Yaskawa INFORM job: OK_R2_O57-69(2)(90,0)_OK_HARDOX.JBI

/JOB
//NAME OK_R2_O57-69(2)(90,0)_OK_HARDOX
///FOLDERNAME X4
//POS
///NPOS 604,604,604,23,0,0
///TOOL 0
///POSTYPE PULSE
///PULSE
C00000=-135424,72899,29147,-3537,85342,3792
C00001=-134013,95021,61136,-4029,77105,4505
C00002=-134047,101087,71818,-4077,73656,4607
C00003=-134047,101216,72822,-4088,73105,4626
C00004=-134047,101094,71866,-4078,73630,4609
C00005=-133936,105187,77198,-4137,72460,4688
C00006=-134047,101094,71866,-4078,73630,4609
C00007=-133891,92563,58880,-4064,77236,4542
C00008=-133627,85963,47659,-4101,80754,4516
C00009=-133192,78294,50454,-10127,76922,11696
C00010=-133849,85255,61933,-10093,73405,11757
C00011=-135353,87618,67605,-9788,70974,11422
C00012=-135353,87997,69106,-9827,70255,11481
C00013=-135353,87618,67605,-9788,70974,11422
C00014=-135153,93739,75342,-9940,69404,11624
C00015=-135353,87618,67605,-9788,70974,11422
C00016=-133639,83161,60388,-10158,73308,11840
C00017=-132974,76301,49087,-10194,76769,11784
C00018=-129415,62996,33414,-11066,79991,12732
C00019=-98130,32671,61537,-45409,44339,32891
C00020=-100023,41688,73231,-46965,41628,33506
C00021=-100756,49088,84228,-49401,39255,34803
C00022=-100756,52120,89278,-50881,38240,35655
C00023=-100756,49088,84228,-49401,39255,34803
C00024=-101219,51120,86580,-49709,38764,34882
C00025=-100756,49088,84228,-49401,39255,34803
C00026=-97195,31965,62320,-46227,44186,33575
C00027=-75566,-2034,22500,-42402,86688,50389
C00028=-92276,-18388,7402,-33699,73725,46550
C00029=-92276,-17400,9548,-33822,73042,46763
C00030=-92276,-17933,8393,-33755,73407,46648
C00031=-120131,-32698,-12117,4829,66200,34356
C00032=-120131,-32114,-10702,4851,65630,34332
C00033=-120989,-32117,-10704,5006,65680,34020
C00034=-120131,-32114,-10702,4851,65630,34332
C00035=-120131,-38085,-26806,4645,72450,34604
C00036=-99101,-76935,-92016,-31014,74911,20401
C00037=-52587,-144740,-101483,-60524,64363,-65274
C00038=-46989,-65360,-59229,-62781,73103,-77672
C00039=-56832,-65466,-56421,-59287,64983,-77772
C00040=-57148,-65688,-55453,-59188,64110,-77279
C00041=-55649,-62097,-53047,-61106,66880,-78547
C00042=-57237,-59710,-51792,-60669,66110,-79037
C00043=-56277,-61326,-53166,-60831,66721,-78866
C00044=-55441,-62561,-53810,-61057,67127,-78609
C00045=-56207,-63985,-54541,-61032,66503,-78630
C00046=-55438,-62578,-53813,-61060,67126,-78606
C00047=-51973,-62323,-54701,-62406,69323,-78001
C00048=-48054,-62529,-57040,-62601,72472,-77896
C00049=-29811,-70761,-60283,-66780,94863,-53671
C00050=-30965,-22538,-31531,-67696,97011,-56857
C00051=-55044,-42598,-44870,-68563,88788,-43678
C00052=-56249,-45120,-46406,-68472,87844,-43687
C00053=-57925,-45354,-44812,-68371,86292,-43442
C00054=-57925,-45174,-43802,-68390,86084,-43215
C00055=-57925,-45354,-44812,-68371,86292,-43442
C00056=-59167,-45210,-44726,-68282,85469,-43617
C00057=-57925,-45354,-44812,-68371,86292,-43442
C00058=-55819,-44223,-45863,-68504,88181,-43684
C00059=-44722,-31045,-43816,-69927,97696,-44632
C00060=-43071,-26445,-40665,-70170,98951,-44614
C00061=-127706,-49493,-81773,19458,97242,-49666
C00062=-127020,6423,-39070,7004,99714,-51816
C00063=-127020,5137,-37554,6966,98131,-51906
C00064=-128416,4382,-35850,7239,96821,-52416
C00065=-128416,3847,-35017,7224,96041,-52460
C00066=-128416,4148,-35496,7233,96488,-52435
C00067=-130041,4566,-35136,7580,96617,-52937
C00068=-129924,4205,-34639,7545,96120,-52933
C00069=-129457,4078,-34747,7447,96082,-52788
C00070=-130190,4712,-35256,7614,96778,-52976
C00071=-128966,36168,-17458,7491,101844,-52285
C00072=-149392,-6912,-25974,9982,75562,-31317
C00073=-149173,-488,-12666,10148,70714,-31647
C00074=-149173,-326,-10897,10208,69722,-31733
C00075=-149173,-394,-11578,10184,70101,-31701
C00076=-148123,2416,-9216,9823,69962,-31333
C00077=-149173,-394,-11578,10184,70101,-31701
C00078=-152478,4885,-6741,15795,72623,-37698
C00079=-151455,3828,-7649,15488,72442,-37350
C00080=-152478,4560,-12614,15554,75946,-37261
C00081=-146445,-24647,-43161,13522,78564,-34847
C00082=-131268,-45047,-56509,8633,74300,53297
C00083=-142507,25021,6402,32310,105830,54923
C00084=-142507,25105,7931,32155,105064,54695
C00085=-142507,25067,7336,32214,105361,54783
C00086=-144899,27115,9325,31955,106116,54020
C00087=-144899,27165,10051,31882,105756,53914
C00088=-143964,26333,9240,31989,105467,54213
C00089=-144899,27115,9325,31955,106116,54020
C00090=-139799,26044,8286,32411,104272,55572
C00091=-139799,26086,8928,32350,103953,55476
C00092=-140218,24332,7231,32337,104232,55386
C00093=-139845,24485,5469,32557,105080,55794
C00094=-133821,6451,-11055,33047,103540,57803
C00095=-133821,6495,-9064,32866,102523,57496
C00096=-133821,6476,-9598,32913,102793,57577
C00097=-132525,9567,-6887,32955,102227,57935
C00098=-132525,9588,-6343,32910,101953,57853
C00099=-133066,7796,-7920,32894,102203,57708
C00100=-133013,8554,-8607,33013,102871,57931
C00101=-134496,-11545,-24055,37394,79049,50318
C00102=-128731,-14923,-26642,36062,76491,51870
C00103=-127482,-15460,-24018,36014,74425,51702
C00104=-127482,-15304,-22595,36136,73774,51482
C00105=-127482,-15363,-23111,36090,74009,51562
C00106=-129060,-19650,-26295,36507,74476,51047
C00107=-129060,-19568,-25628,36564,74177,50944
C00108=-128523,-17977,-24457,36422,74028,51123
C00109=-129540,-19245,-27224,36505,75313,51130
C00110=-136115,2071,-10391,37882,78617,49479
C00111=-137580,2242,-9921,38197,79097,49024
C00112=-137580,2375,-8533,38282,78470,48799
C00113=-137580,2298,-9294,38235,78811,48922
C00114=-139070,-1458,-12440,38519,79473,48520
C00115=-139070,-1365,-11538,38571,79071,48374
C00116=-138460,140,-10285,38458,78803,48541
C00117=-138988,-820,-13903,38388,80409,48895
C00118=-141740,13451,-1511,38926,81398,48075
C00119=-142514,14144,562,39136,81023,47605
C00120=-142514,14274,1799,39195,80477,47404
C00121=-142514,14207,1180,39164,80748,47504
C00122=-144026,10774,-1912,39404,81538,47142
C00123=-144026,10851,-1183,39436,81218,47023
C00124=-143517,12181,9,39358,80948,47144
C00125=-143717,11422,-2918,39282,82143,47501
C00126=-140568,19291,1223,17454,68729,44783
C00127=-141248,20501,3331,17792,68230,44452
C00128=-141248,20564,4327,17861,67675,44366
C00129=-141248,20543,3999,17838,67857,44394
C00130=-142986,16313,57,18468,68479,43839
C00131=-142986,16348,619,18508,68167,43788
C00132=-142176,18240,2371,18214,67887,44048
C00133=-142876,17282,-1215,18280,69673,44071
C00134=-131494,-80468,-98534,7816,92108,-53678
C00135=-52065,-14099,-27709,-42253,108676,27596
C00136=-76671,-130461,-121705,-35735,90710,50834
C00137=-94829,-93442,-100428,-28991,96183,47377
C00138=-110716,-92055,-82664,-19311,98038,51285
C00139=-114275,-93352,-80055,-19461,95045,50478
C00140=-118122,-92212,-76367,-19656,92534,49497
C00141=-118129,-91398,-74848,-19645,92046,49575
C00142=-118122,-92212,-76367,-19656,92534,49497
C00143=-119808,-92271,-76389,-19753,92113,48959
C00144=-118122,-92212,-76367,-19656,92534,49497
C00145=-114499,-91094,-78376,-19482,95112,50387
C00146=-110992,-89821,-80983,-19339,98080,51178
C00147=-124454,-89651,-86550,11137,94998,-69701
C00148=-122569,-92184,-83910,11067,91866,-69331
C00149=-120652,-93960,-80852,11027,88857,-68936
C00150=-120652,-93520,-79457,11027,88237,-68992
C00151=-120652,-93960,-80852,11027,88857,-68936
C00152=-120650,-97396,-81866,11026,87737,-69033
C00153=-120652,-93960,-80852,11027,88857,-68936
C00154=-118161,-93768,-80427,10994,88357,-68121
C00155=-120652,-93960,-80852,11027,88857,-68936
C00156=-120037,-91891,-82714,11032,90945,-68539
C00157=-121981,-89592,-85452,11099,94026,-68936
C00158=-122005,-89480,-97857,11363,101580,-68254
C00159=-122005,-89427,-98101,11372,101754,-68238
C00160=-119094,-95812,-115555,-4544,90851,-20867
C00161=-116502,-111480,-109655,-18779,62868,21987
C00162=-119472,-101923,-104261,-17094,63743,20698
C00163=-121534,-96097,-100090,-16016,63743,19914
C00164=-121534,-96194,-98882,-16123,62979,20025
C00165=-112336,-84014,-94514,-26506,72534,27449
C00166=-114298,-84401,-94682,-25743,71847,26864
C00167=-121534,-96097,-100090,-16016,63743,19914
C00168=-121514,-92242,-98700,-15883,64832,19765
C00169=-121534,-96097,-100090,-16016,63743,19914
C00170=-119823,-101836,-103002,-17025,62972,20682
C00171=-116876,-111303,-108368,-18711,62117,21969
C00172=-126032,-109701,-108999,21760,66785,-27050
C00173=-122513,-101468,-103921,20079,66940,-25677
C00174=-121483,-94377,-99419,19507,67520,-25186
C00175=-121483,-94509,-98158,19621,66724,-25324
C00176=-121483,-94377,-99419,19507,67520,-25186
C00177=-119206,-94355,-99408,18489,67008,-24418
C00178=-121483,-94377,-99419,19507,67520,-25186
C00179=-121468,-91005,-98354,19362,68535,-25006
C00180=-121483,-94377,-99419,19507,67520,-25186
C00181=-124810,-108862,-107603,21303,66070,-26716
C00182=-126981,-112864,-109311,24940,61360,-29729
C00183=-123200,-104180,-104415,22777,61614,-28126
C00184=-121230,-90686,-98732,21152,64298,-26805
C00185=-121230,-90968,-97120,21351,63235,-27013
C00186=-121230,-90806,-98119,21226,63888,-26884
C00187=-118688,-90754,-98099,19926,63280,-26013
C00188=-121230,-90721,-98563,21173,64184,-26826
C00189=-121211,-84894,-96124,20922,65577,-26553
C00190=-121230,-90686,-98732,21152,64298,-26805
C00191=-121413,-93580,-100796,21282,64141,-26906
C00192=-124847,-101623,-105736,23178,64029,-28268
C00193=-120616,-95755,-103879,23668,64726,-45447
C00194=-120621,-89459,-99052,23623,64971,-45396
C00195=-102398,-78806,-99215,-137,71874,-40792
C00196=-120614,-97387,-102466,23992,63157,-45792
C00197=-122354,-96256,-100860,24938,63287,-46459
C00198=-99477,-102621,-105563,-1650,63574,-39713
C00199=-93449,-138180,-112622,-5538,49931,-36849
C00200=-85999,-163182,-115201,-11989,39587,-32297
C00201=-96470,-180165,-126119,-4784,36529,-37522
C00202=-120616,-95173,-105764,23303,89544,-42444
C00203=-107191,-96001,-89285,21702,28532,-58770
C00204=-107187,-93630,-79997,25295,24388,-60561
C00205=-107188,-92928,-77886,26213,23539,-61010
C00206=-112362,-77289,-77026,28293,40281,-63318
C00207=-107081,-94020,-78768,26067,23489,-60939
C00208=-108911,-93070,-77209,29349,23678,-62538
C00209=-100555,-91608,-91171,7273,48196,-53989
C00210=-102645,-104114,-96524,14611,51707,-64227
C00211=-108915,-55552,-83371,19664,91458,-62056
C00212=-110657,-50226,-86705,20295,96355,-61815
C00213=-107202,-93991,-108886,21178,109925,-43661
C00214=-120660,-73953,-111348,177,99224,835
C00215=-120616,-96234,-101081,-23944,56754,46777
C00216=-120615,-96493,-97034,-24670,54353,47364
C00217=-120614,-96447,-94923,-25055,53191,47662
C00218=-125343,-63714,-87611,-17170,75461,41479
C00219=-118876,-96360,-94049,-26267,53277,48431
C00220=-120612,-97621,-95709,-25094,53083,47691
C00221=-124024,-105215,-109245,-22308,82546,38090
C00222=-123496,-104488,-108175,-22872,85665,42107
C00223=-120617,-94319,-107453,-23464,90858,42123
C00224=-120617,-92878,-109780,-23521,92858,41729
C00225=-120619,-86141,-115603,-23930,99335,40429
C00226=-120619,-89012,-115558,8782,73464,77384
C00227=-120618,-92353,-112869,8941,70132,77138
C00228=-120618,-93422,-111698,9011,68877,77043
C00229=-120616,-94109,-113157,8979,69414,77085
C00230=-120318,-89311,-110489,8778,70198,77244
C00231=-120618,-93688,-111329,9132,68044,76969
C00232=-120618,-93957,-110924,9216,67187,76884
C00233=-120618,-94299,-110440,9161,65769,76809
C00234=-120618,-94831,-109599,8469,63241,76696
C00235=-120617,-95145,-109027,7071,61401,76664
C00236=-120617,-95217,-108863,5672,60665,76701
C00237=-120618,-93036,-111930,4923,63538,76718
C00238=-120618,-92960,-112001,4009,63579,76743
C00239=-120618,-92691,-112274,2433,64167,76800
C00240=-120618,-92166,-112798,840,65602,76863
C00241=-120618,-91419,-113490,-342,67708,76910
C00242=-120619,-90739,-114068,-878,69589,76936
C00243=-120619,-89701,-115007,-939,71612,76812
C00244=-120619,-88814,-115609,-873,73870,76855
C00245=-120619,-87740,-116270,-151,76574,76959
C00246=-120619,-86987,-116700,1182,78540,77121
C00247=-120619,-86782,-116823,2462,79296,77267
C00248=-120619,-90672,-114378,3278,75949,77117
C00249=-120619,-90769,-114313,4130,75889,77177
C00250=-120619,-91109,-114056,5597,75252,77256
C00251=-120618,-91719,-113544,7101,73764,77286
C00252=-120618,-92472,-112836,8259,71637,77242
C00253=-120618,-92872,-112418,8666,70405,77193
C00254=-120618,-93168,-112034,8862,69621,77111
C00255=-120618,-93422,-111698,9011,68877,77043
C00256=-120618,-92353,-112869,8941,70132,77138
C00257=-120619,-89012,-115558,8782,73464,77384
C00258=-120595,-119438,-127420,-8829,91162,8830
C00259=-129025,-103888,-99333,21372,86937,-54976
C00260=-120613,-94952,-86848,20336,81911,-52813
C00261=-120613,-94069,-83278,20415,80272,-53091
C00262=-106596,-117430,-87528,9818,57368,-33279
C00263=-120519,-95091,-83551,20421,79912,-53118
C00264=-122104,-92396,-81537,20633,80446,-53604
C00265=-112247,-111615,-87090,12951,66121,-41348
C00266=-120242,-93380,-81431,16167,85346,-56835
C00267=-120729,-92389,-78218,16226,84033,-57178
C00268=-121550,-94001,-78799,15119,86025,-61641
C00269=-122325,-96218,-79481,13215,89152,-68718
C00270=-120612,-93818,-82398,13271,91824,-67835
C00271=-120613,-94827,-86367,13308,93699,-67633
C00272=-120614,-96085,-95173,13466,98348,-67128
C00273=-120625,-105302,-100360,13404,96846,-67297
C00274=-102872,-120945,-93289,-41313,52454,35552
C00275=-111052,-89986,-73102,-36259,51528,31574
C00276=-114360,-89865,-71590,-35102,49434,30694
C00277=-117529,-82976,-67958,-32873,49251,29097
C00278=-113966,-89555,-70876,-35431,49366,30932
C00279=-115650,-91167,-72721,-34446,48930,30213
C00280=-116153,-87173,-73787,-30474,57370,33009
C00281=-115134,-90585,-78921,-28213,65812,37618
C00282=-114816,-93273,-83340,-25850,75230,43378
C00283=-115191,-85090,-71836,-25015,76673,46996
C00284=-114907,-96450,-75026,-24463,77444,52852
C00285=-115702,-94689,-74701,-23512,87260,62633
C00286=-112822,-91718,-77371,-23458,91001,62960
C00287=-109330,-92095,-80656,-23399,93677,63722
C00288=-110759,-94815,-97268,-24043,101385,61640
C00289=-25230,-87703,-86789,-41333,106155,-71905
C00290=-55862,19660,17206,-68346,89547,-53836
C00291=-59225,37567,25812,-69215,105770,-42705
C00292=-67658,42850,42597,-68102,97125,-40508
C00293=-69543,42635,44538,-68129,95346,-40204
C00294=-67599,42910,43858,-67984,96867,-40179
C00295=-68366,42138,41747,-68199,96713,-40671
C00296=-69537,42554,44453,-68130,95355,-40208
C00297=-69167,26414,28126,-68889,91591,-41841
C00298=-69430,8343,11443,-69273,87154,-43187
C00299=-70467,-11089,-4532,-69437,78929,-44678
C00300=-70464,-3151,1747,-68553,83829,-57137
C00301=-68177,-4212,-1280,-68454,85880,-57398
C00302=-65815,-3605,-3490,-68417,88124,-57797
C00303=-46513,-27715,-22241,-69125,80479,-38621
C00304=-7625,-19791,-74194,-84461,116832,-51132
C00305=-98528,-26744,-48644,-33463,55012,-18344
C00306=-113253,15209,27106,-3834,50657,3406
C00307=-113409,21623,32322,-3755,50736,3338
C00308=-112510,30954,47444,-4478,46281,3921
C00309=-113472,24070,39362,-3899,47665,3430
C00310=-113579,25546,39455,-3805,48359,3355
C00311=-112547,30896,47385,-4459,46286,3903
C00312=-113092,30984,47541,-6567,46499,5785
C00313=-107982,35826,53096,-19952,49307,15286
C00314=-107346,38752,56151,-24065,51859,19797
C00315=-102444,58818,79888,-34511,57818,35075
C00316=-101044,76619,103296,-39601,59307,41475
C00317=-99948,73081,91706,-37976,69105,42304
C00318=-99205,63215,84174,-37575,62603,39615
C00319=-97180,56339,73463,-36771,65900,39269
C00320=-108272,10166,23438,-3323,45242,19316
C00321=-109103,10218,12469,-2549,51979,18742
C00322=-99879,30934,32617,-21980,59339,34187
C00323=-99785,30090,30578,-21838,60128,34061
C00324=-99052,29053,30612,-22206,59809,34434
C00325=-101543,26260,28122,-21325,59243,33514
C00326=-98482,32149,35009,-29284,63220,41247
C00327=-92009,66840,89116,-42947,61850,57046
C00328=-89877,62120,80876,-42077,64804,56709
C00329=-70258,15873,38394,-48666,102593,69187
C00330=-68816,9929,45318,-53577,93501,68972
C00331=-74323,28982,63484,-55349,89726,68465
C00332=-74758,1474,21309,-45746,90270,65676
C00333=-98607,12568,39814,52966,86937,78252
C00334=-98596,22842,59344,53301,82774,75788
C00335=-96296,21421,60413,54092,80731,75703
C00336=-95348,20952,60953,54433,79893,75663
C00337=-96117,19164,58324,54129,80713,75783
C00338=-95662,23434,63388,54370,79922,75521
C00339=-95503,21312,61702,54422,79811,75531
C00340=-92574,18445,54645,48983,79889,68258
C00341=-91800,17848,53101,47601,79897,67557
C00342=-92530,17999,51917,47342,80806,67673
C00343=-94302,18640,49262,46764,83033,67943
C00344=-79003,18324,29303,31626,94586,4503
C00345=-64136,40618,57122,29721,84915,83830
C00346=-62802,39067,58740,29997,82892,83805
C00347=-62255,38544,59506,30121,82059,83791
C00348=-62254,37103,56589,30066,82978,84033
C00349=-62821,40643,61741,30049,81995,83562
C00350=-59984,48909,70165,26795,84201,83115
C00351=-59410,69261,96131,25367,86084,74959
C00352=-59404,69357,96256,25356,86081,74939
C00353=-59713,70793,96681,25260,86600,74945
C00354=-60461,74839,98386,25037,87745,74932
C00355=-60470,59585,70460,25309,96249,76737
C00356=-66845,10330,41939,25249,64720,33768
C00357=-66816,16396,52426,25952,61688,33052
C00358=-66804,19142,57057,26292,60387,32730
C00359=-66058,20615,58344,26298,60142,32956
C00360=-66868,17219,53699,26035,61378,32955
C00361=-66973,19658,57552,26302,60399,32669
C00362=-66985,16895,52895,25961,61707,32992
C00363=-67015,10800,42362,25255,64752,33711
C00364=-98181,31350,57269,53093,86032,77938
C00365=-96082,29267,57446,53647,84171,77916
C00366=-95219,28523,57622,53885,83405,77901
C00367=-95917,26905,55160,53675,84199,78019
C00368=-95506,31088,60230,53837,83386,77740
C00369=-95359,28788,58259,53869,83329,77779
C00370=-92697,26913,52373,48450,83827,70215
C00371=-91994,26523,51069,47073,83939,69440
C00372=-92656,26997,50292,46905,84772,69532
C00373=-94270,28412,48618,46533,86809,69749
C00374=-79891,40483,43632,25605,98381,-17488
C00375=-64421,55368,61348,15926,95442,-62339
C00376=-63205,52871,61672,16144,93779,-62133
C00377=-62708,51961,61917,16235,93087,-62052
C00378=-62707,50761,59239,16263,94078,-61920
C00379=-63223,54241,64482,16113,92796,-62269
C00380=-60236,62044,73663,12795,94061,-63101
C00381=-59090,69141,83012,10500,94867,-70833
C00382=-59083,69182,83067,10487,94869,-70851
C00383=-59379,71028,84054,10408,95242,-70919
C00384=-60098,76023,87068,10213,96031,-71094
C00385=-60107,66003,66038,10511,103704,-70448
C00386=-66860,35146,61423,22993,49349,53528
C00387=-66834,42827,74568,24499,45535,52525
C00388=-66824,46660,80883,25305,43786,52015
C00389=-66175,48781,83167,25255,43321,52183
C00390=-66880,43946,76304,24713,45097,52378
C00391=-66970,47398,81721,25407,43702,51920
C00392=-66981,43500,75311,24586,45473,52438
C00393=-67007,35727,62031,23060,49318,53454
C00394=-87565,40229,55167,37616,76398,68031
C00395=-104252,61764,84947,51561,88394,76219
C00396=-102517,58043,82852,52038,87086,76344
C00397=-101804,56689,82195,52237,86527,76380
C00398=-102435,54601,78919,52052,87454,76595
C00399=-101993,60636,86873,52209,86091,76036
C00400=-101932,57147,83104,52210,86393,76238
C00401=-99529,53434,74771,46937,87155,68655
C00402=-98895,52660,72970,45595,87312,67859
C00403=-99433,53501,72680,45467,88010,67934
C00404=-100745,55861,72292,45181,89689,68100
C00405=-89942,52639,54543,22757,100290,-22350
C00406=-84530,60242,66965,10989,97828,-69052
C00407=-83700,56528,65849,11170,96516,-68885
C00408=-83359,55133,65530,11245,95959,-68819
C00409=-83358,53843,62725,11276,97003,-68723
C00410=-83705,58033,68848,11139,95464,-68982
C00411=-80399,62193,73871,7256,96460,-69699
C00412=-78998,67441,80988,4366,97017,-77318
C00413=-78990,67470,81028,4351,97018,-77335
C00414=-79114,69587,82331,4315,97310,-77366
C00415=-79414,75293,86196,4226,97877,-77446
C00416=-79422,65472,65446,4368,105580,-77179
C00417=-80352,27457,54566,26195,53383,48637
C00418=-80356,27473,54581,26196,53382,48635
C00419=-80357,27479,54587,26196,53382,48634
C00420=-79589,28666,55655,26054,53112,48894
C00421=-80424,25883,51570,25884,54338,48863
C00422=-80357,27479,54587,26196,53382,48634
C00423=-80356,27473,54581,26196,53382,48635
C00424=-80352,27458,54566,26195,53383,48637
C00425=-110061,-17560,-36552,26636,92274,45980
C00426=-111839,-83491,-103870,27371,99587,47031
C00427=-38426,-40229,-52385,-46753,77455,-20722
C00428=-20805,-37224,-43776,-64442,70782,-24410
C00429=-53615,-60479,-29767,-71413,48188,-35364
C00430=-53622,-60473,-29764,-71411,48184,-35366
C00431=-53625,-60471,-29763,-71411,48182,-35366
C00432=-52450,-61746,-30400,-71683,48877,-35041
C00433=-53622,-61330,-31549,-70858,48414,-35743
C00434=-53667,-60425,-29740,-73440,59962,-39458
C00435=-53705,-60384,-29719,-74506,70698,-55233
C00436=-53706,-60382,-29718,-74560,71274,-55582
C00437=-53707,-60381,-29717,-74560,71274,-55582
C00438=-53710,-60377,-29715,-74560,71273,-55583
C00439=-53701,-60384,-29719,-74560,71278,-55581
C00440=-66706,-54450,-33709,-25643,46200,-1067
C00441=-66709,-54445,-33707,-25641,46199,-1069
C00442=-65806,-56035,-34565,-26242,46218,-617
C00443=-67582,-55929,-35261,-25089,46110,-1484
C00444=-66709,-54446,-33707,-25645,46199,-1067
C00445=-66709,-54446,-33707,-25645,46199,-1067
C00446=-66709,-54447,-33708,-25641,46199,-1069
C00447=-66706,-54452,-33711,-25643,46199,-1067
C00448=-56114,-41526,-33189,-36880,64877,1074
C00449=-62492,-26274,-11536,-67617,51989,-49416
C00450=-67015,-30786,-7269,-70211,42036,-48662
C00451=-67021,-30777,-7263,-70209,42033,-48664
C00452=-67024,-30773,-7260,-70208,42031,-48665
C00453=-67025,-30771,-7259,-70208,42030,-48665
C00454=-66245,-32305,-8266,-70488,42489,-48421
C00455=-67024,-31573,-9128,-69442,42305,-49131
C00456=-67037,-30747,-7244,-72021,47713,-46269
C00457=-67060,-30703,-7215,-71923,58333,-61620
C00458=-67063,-30697,-7211,-72128,59825,-62445
C00459=-67063,-30696,-7209,-72128,59824,-62445
C00460=-67065,-30691,-7207,-72128,59824,-62445
C00461=-67053,-30709,-7218,-72128,59831,-62443
C00462=-67069,40537,9457,-57195,76262,-35492
C00463=-67067,40166,11985,-57536,75289,-34802
C00464=-67066,40064,13042,-57682,74899,-34523
C00465=-66577,38326,11242,-57768,75308,-34517
C00466=-67065,40169,11907,-57527,75318,-34822
C00467=-67072,40075,13170,-59772,79795,-32172
C00468=-67078,40614,25191,-75815,82535,-42307
C00469=-67079,40861,26780,-77445,83659,-42995
C00470=-67080,40685,25622,-77394,83811,-43275
C00471=-67085,40340,22831,-77277,84191,-43970
C00472=-67090,40073,14255,-76963,85485,-46282
C00473=-90837,-14160,-23602,-46112,79870,29092
C00474=-94881,-86110,-91503,-45134,79065,22948
C00475=-94881,-86110,-91503,-45134,79065,22948
C00476=-94881,-86110,-91503,-45134,79065,22948
C00477=-64023,-117945,-92652,-70836,68337,-59810
C00478=-77839,-63283,-64145,-64455,63318,-66711
C00479=-80052,-65654,-65354,-64094,61673,-66872
C00480=-91542,-73752,-69062,-57934,49878,-61172
C00481=-80955,-66618,-66084,-63874,61070,-67008
C00482=-80000,-68279,-65664,-64663,61180,-66324
C00483=-91387,-73280,-68839,-57922,50030,-61186
C00484=-100914,-85483,-74196,-43298,32083,-69038
C00485=-93618,-76672,-70228,-47057,37292,-67140
C00486=-87612,-64529,-64461,-48733,42323,-66403
C00487=-94575,-77342,-71004,-49651,37504,-40583
C00488=-95005,-77606,-71124,-49413,37228,-40705
C00489=-25543,-37396,-56331,-69239,85891,-31897
C00490=-172418,-62024,-69195,63943,69139,25706
C00491=-192822,-61773,-75094,68063,83874,24345
C00492=-147462,40071,30365,69170,75532,19593
C00493=-147457,40119,30415,69171,75526,19591
C00494=-147456,40127,30423,69171,75525,19590
C00495=-147721,37841,28052,69134,75813,19681
C00496=-148042,40615,30212,69143,76066,19681
C00497=-147457,40126,30423,69172,75522,19590
C00498=-147457,40126,30423,69172,75522,19590
C00499=-147457,40125,30422,69171,75526,19590
C00500=-147458,40117,30413,69171,75527,19591
C00501=-147460,40097,30392,69171,75529,19592
C00502=-134071,6209,-12454,63265,71876,23505
C00503=-134070,6228,-12438,63265,71875,23505
C00504=-134070,6235,-12431,63265,71875,23505
C00505=-134229,4110,-14261,63296,71992,23494
C00506=-134787,6570,-12855,63330,72532,23573
C00507=-134070,6235,-12432,63265,71872,23505
C00508=-134070,6235,-12432,63265,71872,23505
C00509=-134071,6233,-12433,63265,71876,23505
C00510=-134071,6226,-12439,63265,71876,23505
C00511=-134072,6208,-12455,63265,71877,23505
C00512=-134072,6180,-12479,63265,71877,23505
C00513=-130462,-25122,-37090,45275,45470,33351
C00514=-132886,-107940,-72929,67003,34868,20711
C00515=-175339,-34674,-82182,59494,83195,32396
C00516=-136096,14126,-32620,12825,85534,21552
C00517=-129268,63666,34345,-8258,78331,9264
C00518=-134681,92240,52646,-816,80365,910
C00519=-132653,94106,63405,6765,75468,-3487
C00520=-132876,98805,66718,-7260,76138,8167
C00521=-132758,95444,63654,-7290,76306,8197
C00522=-134693,106943,79821,5995,71756,-2669
C00523=-133635,106832,79602,3484,71508,162
C00524=-131960,102921,75089,-426,70802,5631
C00525=-130942,105589,75064,-6359,73995,10618
C00526=-131542,109137,74044,-11980,78923,13777
C00527=-129355,125982,76686,-9729,88276,13921
C00528=-127789,121294,71761,-15545,88654,13573
C00529=-127928,122256,73029,-17074,89645,15674
C00530=-128241,121543,71989,-17007,89844,15541
C00531=-129796,115422,63669,-14368,89697,11833
C00532=-130249,115476,63291,-14256,89876,11663
C00533=-129188,109453,52652,-14573,93397,11596
C00534=-127389,117603,65505,-15655,90606,13460
C00535=-137764,37902,26809,9618,64282,22430
C00536=-175415,-47626,-48014,65040,69542,20935
C00537=-132886,-107940,-72929,67003,34868,20711
C00538=-105972,-100304,-88890,7532,75015,-38248
C00539=-160165,-106496,-82005,21656,82129,-62098
C00540=-140609,-94579,-78221,8463,77656,-55534
C00541=-138726,-94535,-76086,8242,76183,-54976
C00542=-163390,-101496,-77356,21709,82707,-63168
C00543=-161792,-103413,-79036,21690,82331,-62654
C00544=-135933,-74368,-67331,7717,80836,-53706
C00545=-133468,-45426,-54020,7292,87230,-52484
C00546=-132807,-44691,-51453,7196,85977,-52334
C00547=-131271,-21709,-36375,6964,88353,-51682
C00548=-131369,-20934,-44335,7010,93621,-51422
C00549=-131369,-20934,-44335,7010,93621,66180
C00550=-144527,-21077,-33351,28595,78219,62582
C00551=-141662,-29032,-35117,26435,70731,67420
C00552=-141636,-28849,-34992,26424,70738,67431
C00553=-141636,-28849,-34992,26424,70738,67431
C00554=-141058,-3119,-19308,25775,87573,66314
C00555=-137634,17841,-2515,22739,98686,69533
C00556=-136794,15937,-4297,22735,98567,69816
C00557=-135468,13055,-6959,22721,98352,70259
C00558=-124155,-6946,-23990,22264,95502,73827
C00559=-124092,-3412,-25453,22421,98006,74321
C00560=-141014,2861,-12124,36786,79556,66317
C00561=-139301,5079,-6063,36704,76730,66076
C00562=-139384,4271,-6757,36720,76775,66056
C00563=-139395,3578,-7350,36721,76786,66055
C00564=-139375,2979,-7861,36717,76784,66060
C00565=-139252,2411,-8343,36689,76734,66096
C00566=-139094,1918,-8761,36656,76670,66141
C00567=-138273,63,-10319,36478,76326,66373
C00568=-124702,-23193,-28294,33182,70061,70062
C00569=-125787,-25173,-32450,33220,71783,70141
C00570=-117588,-7377,-27060,-792,74259,70914
C00571=-118143,-3971,-19985,-599,71653,70736
C00572=-118337,-4947,-20776,-528,71638,70668
C00573=-118455,-18119,-27040,-763,60705,70665
C00574=-119252,-27594,-29328,-557,49936,70400
C00575=-122681,-23558,-26502,1731,50293,68913
C00576=-141762,10837,837,13868,52999,60935
C00577=-147205,15689,5640,25604,56460,59753
C00578=-147231,16301,6201,25627,56440,59736
C00579=-147475,14155,1624,25286,58068,60041
C00580=-125492,-45791,-60900,11855,60410,-6355
C00581=-155973,16228,-7521,23092,85783,-46465
C00582=-155545,22569,6657,24866,83301,-50186
C00583=-156114,24235,11083,24511,80804,-49715
C00584=-157855,17121,1644,24703,83284,-49844
C00585=-148516,-1727,-14860,9883,71341,-31357
C00586=-147742,1394,-9472,9715,69559,-31227
C00587=-138592,3455,-7934,-8851,69391,-13105
C00588=-137116,-4730,-20716,-9180,73171,-12868
C00589=-138249,-12129,-32669,-1567,78549,-18356
C00590=-145553,-60948,-35045,47196,66698,-53129
C00591=-117087,2274,-4333,-74835,51753,34811
C00592=-120822,45639,36263,-74296,46580,35142
C00593=-132292,76688,41038,-57812,44611,25328
C00594=-133587,85399,43635,-54635,45518,23471
C00595=-134089,87151,52872,-58446,42500,25922
C00596=-133465,87868,53767,-58981,42776,26187
C00597=-134426,84651,49764,-57666,42643,25479
C00598=-134089,87030,55209,-59870,41700,26787
C00599=-134090,96417,89471,-79265,35490,37858
C00600=-134090,100042,96821,-83028,34997,39924
C00601=-133589,94413,89775,-81024,35602,38850
C00602=-132294,83338,76456,-77824,37058,37121
C00603=3643,-76224,-106676,19950,71810,76872
BC00000=138406,837384,245994
BC00001=138406,837384,245994
BC00002=138406,837384,245994
BC00003=138406,837384,245994
BC00004=138406,837384,245994
BC00005=138406,837384,245994
BC00006=138406,837384,245994
BC00007=138406,837384,245994
BC00008=138406,837384,245994
BC00009=128112,840549,330774
BC00010=128112,840549,330774
BC00011=128112,840549,330774
BC00012=128112,840549,330774
BC00013=128112,840549,330774
BC00014=128112,840549,330774
BC00015=128112,840549,330774
BC00016=128112,840549,330774
BC00017=128112,840549,330774
BC00018=128112,840549,330774
BC00019=111975,837625,420975
BC00020=111975,837625,420975
BC00021=111975,837625,420975
BC00022=111975,837625,420975
BC00023=111975,837625,420975
BC00024=111976,837626,420972
BC00025=111975,837625,420975
BC00026=111975,837625,420975
BC00027=111975,837625,420975
BC00028=111975,837625,420975
BC00029=111975,837625,420975
BC00030=111975,837625,420975
BC00031=111975,837625,420975
BC00032=111975,837625,420975
BC00033=111975,837625,420975
BC00034=111975,837625,420975
BC00035=111975,837625,420975
BC00036=111578,670431,418295
BC00037=342650,733121,86647
BC00038=339628,728489,87096
BC00039=339628,728489,87096
BC00040=339628,728489,87096
BC00041=339628,728489,87096
BC00042=339628,728489,87096
BC00043=339628,728489,87096
BC00044=339628,728489,87096
BC00045=339628,728489,87096
BC00046=339628,728489,87096
BC00047=339628,728489,87096
BC00048=339628,728489,87096
BC00049=369440,735504,90134
BC00050=369440,735504,90134
BC00051=398174,741162,97424
BC00052=398174,745386,78467
BC00053=398174,747075,70884
BC00054=398174,747075,70884
BC00055=398174,747075,70884
BC00056=398174,747075,70884
BC00057=398174,747075,70884
BC00058=398174,744503,70979
BC00059=398174,740279,89936
BC00060=398174,693649,89936
BC00061=309739,685336,89936
BC00062=309739,717578,89936
BC00063=309739,717578,89936
BC00064=309739,717578,89936
BC00065=309739,717578,89936
BC00066=309739,717578,89936
BC00067=309739,717578,89936
BC00068=309739,717578,89936
BC00069=309739,717578,89936
BC00070=309739,717578,89936
BC00071=309739,717578,89936
BC00072=311206,810481,212793
BC00073=311206,810481,212793
BC00074=311206,810481,212793
BC00075=311206,810481,212793
BC00076=311206,810481,212793
BC00077=311206,810481,212793
BC00078=311206,810481,212793
BC00079=311206,810481,212793
BC00080=311206,810481,212793
BC00081=311206,810481,212793
BC00082=311206,810481,212793
BC00083=311206,810481,212791
BC00084=311206,810481,212791
BC00085=311206,810481,212791
BC00086=311206,810481,212791
BC00087=311206,810481,212791
BC00088=311206,810481,212791
BC00089=311206,810481,212791
BC00090=311205,810481,212789
BC00091=311205,810481,212789
BC00092=311205,810481,212789
BC00093=311205,810481,212789
BC00094=311205,810481,212789
BC00095=311205,810481,212789
BC00096=311205,810481,212789
BC00097=311205,810481,212789
BC00098=311205,810481,212789
BC00099=311205,810481,212789
BC00100=311205,810481,212789
BC00101=311205,810481,212789
BC00102=311205,810481,212789
BC00103=311205,810481,212789
BC00104=311205,810481,212789
BC00105=311205,810481,212789
BC00106=311205,810481,212789
BC00107=311205,810481,212789
BC00108=311205,810481,212789
BC00109=311205,810481,212789
BC00110=311205,810481,212789
BC00111=311205,810481,212789
BC00112=311205,810481,212789
BC00113=311205,810481,212789
BC00114=311205,810481,212789
BC00115=311205,810481,212789
BC00116=311205,810481,212789
BC00117=311205,810481,212789
BC00118=311205,810481,212789
BC00119=311205,810481,212789
BC00120=311205,810481,212789
BC00121=311205,810481,212789
BC00122=311205,810481,212789
BC00123=311205,810481,212789
BC00124=311205,810481,212789
BC00125=311205,810481,212789
BC00126=311205,810481,212789
BC00127=311205,810481,212789
BC00128=311205,810481,212789
BC00129=311205,810481,212789
BC00130=311205,810481,212789
BC00131=311205,810481,212789
BC00132=311205,810481,212789
BC00133=311205,810481,212789
BC00134=309739,717578,89936
BC00135=302229,671844,714988
BC00136=365201,715179,1005006
BC00137=376221,744487,992760
BC00138=398174,770458,1075175
BC00139=398174,770458,1075175
BC00140=398174,770458,1075175
BC00141=398174,770458,1075175
BC00142=398174,770458,1075175
BC00143=398174,770458,1075175
BC00144=398174,770458,1075175
BC00145=398174,770458,1075175
BC00146=398174,770458,1075175
BC00147=395964,766843,1075175
BC00148=395964,766843,1075175
BC00149=395964,766843,1075175
BC00150=395964,766843,1075175
BC00151=395964,766843,1075175
BC00152=395964,766843,1075175
BC00153=395964,766843,1075175
BC00154=395964,766843,1075175
BC00155=395964,766843,1075175
BC00156=395964,766843,1075175
BC00157=395964,766843,1075175
BC00158=395964,766843,1075175
BC00159=395964,766843,1075175
BC00160=340614,815508,1075175
BC00161=291315,858852,1075175
BC00162=291315,858852,1075175
BC00163=291315,858852,1075175
BC00164=291315,858852,1075175
BC00165=291314,858852,1075172
BC00166=291315,858852,1075175
BC00167=291315,858852,1075175
BC00168=291315,858852,1075175
BC00169=291315,858852,1075175
BC00170=291315,858852,1075175
BC00171=291315,858852,1075175
BC00172=261388,857545,1075175
BC00173=261388,857545,1075175
BC00174=261388,857545,1075175
BC00175=261388,857545,1075175
BC00176=261388,857545,1075175
BC00177=261388,857545,1075175
BC00178=261388,857545,1075175
BC00179=261388,857545,1075175
BC00180=261388,857545,1075175
BC00181=261388,857545,1075175
BC00182=307762,841902,1075175
BC00183=307762,841902,1075175
BC00184=307762,841902,1075175
BC00185=307762,841902,1075175
BC00186=307762,841902,1075175
BC00187=307762,841902,1075175
BC00188=307762,841902,1075175
BC00189=307762,841902,1075175
BC00190=307762,841902,1075175
BC00191=307762,841902,1075175
BC00192=307762,841902,1075175
BC00193=295805,844282,1075175
BC00194=301244,847949,1075175
BC00195=301245,847950,1075171
BC00196=303420,849415,1075175
BC00197=303420,849415,1075175
BC00198=301245,847950,1075171
BC00199=301245,847950,1075171
BC00200=301245,847950,1075171
BC00201=301245,847950,1075171
BC00202=292414,841371,1075175
BC00203=232606,821958,1075175
BC00204=232627,821961,1075175
BC00205=237648,826895,1075175
BC00206=239656,828868,1075175
BC00207=239656,828868,1075175
BC00208=239656,828868,1075175
BC00209=236217,842775,1075175
BC00210=236217,842775,1075175
BC00211=236217,842775,1075175
BC00212=236217,842775,1075175
BC00213=235448,917179,1075175
BC00214=281175,871070,1075175
BC00215=310701,846914,1075175
BC00216=310711,846915,1075175
BC00217=305421,851150,1075175
BC00218=305421,851150,1075175
BC00219=303304,852843,1075175
BC00220=303304,852843,1075175
BC00221=309181,898740,1075175
BC00222=309191,897098,1075175
BC00223=311453,893904,1075175
BC00224=317069,892657,1075175
BC00225=317048,892655,1075175
BC00226=38661,866681,1075175
BC00227=39338,869210,1075175
BC00228=39608,870221,1075175
BC00229=39608,870221,1075175
BC00230=39608,870221,1075175
BC00231=44180,868724,1075175
BC00232=49942,867043,1075175
BC00233=50951,865571,1075175
BC00234=53196,863119,1075175
BC00235=56428,861533,1075175
BC00236=59256,861216,1075175
BC00237=64296,880759,1075175
BC00238=66009,881082,1075175
BC00239=68741,882049,1075175
BC00240=71304,883797,1075175
BC00241=72987,886132,1075175
BC00242=73378,888140,1075175
BC00243=51598,893084,1075175
BC00244=50729,895319,1075175
BC00245=48626,897836,1075175
BC00246=45460,899499,1075175
BC00247=42639,899847,1075175
BC00248=37245,880361,1075175
BC00249=35524,880029,1075175
BC00250=32792,879014,1075175
BC00251=30275,877177,1075175
BC00252=28702,874753,1075175
BC00253=28653,873335,1075175
BC00254=35101,871622,1075175
BC00255=39608,870221,1075175
BC00256=39338,869210,1075175
BC00257=38661,866681,1075175
BC00258=340562,849962,1075175
BC00259=386069,767337,1075175
BC00260=386069,767337,1075175
BC00261=391133,767369,1075175
BC00262=393157,767381,1075161
BC00263=393158,767383,1075175
BC00264=393158,767383,1075175
BC00265=394705,769972,1075166
BC00266=398174,775779,1075175
BC00267=389915,761514,1075175
BC00268=392098,765315,1075171
BC00269=395638,771477,1075175
BC00270=394397,772528,1075175
BC00271=391293,775155,1075175
BC00272=391272,775152,1075175
BC00273=391272,775152,1075175
BC00274=398174,746294,1075175
BC00275=398174,746296,1075175
BC00276=398174,751973,1075175
BC00277=398174,754243,1075175
BC00278=398174,754243,1075175
BC00279=398174,754243,1075175
BC00280=398174,764099,1075175
BC00281=398174,775069,1075175
BC00282=398174,788401,1075175
BC00283=398174,744649,1075175
BC00284=398174,752334,1075175
BC00285=398174,767932,1075175
BC00286=398174,768722,1075175
BC00287=398174,770697,1075175
BC00288=398174,767021,1075175
BC00289=305826,673381,1075175
BC00290=398174,694226,160353
BC00291=398174,710712,168186
BC00292=398174,710712,168186
BC00293=398174,710712,168186
BC00294=398174,710712,168186
BC00295=398174,710712,168186
BC00296=398174,710712,168186
BC00297=398174,710712,168186
BC00298=398174,710712,168186
BC00299=398174,710712,168186
BC00300=398174,710712,168186
BC00301=398174,710712,168186
BC00302=398174,710712,168186
BC00303=398174,694226,160353
BC00304=7965,694226,160353
BC00305=88425,773491,458335
BC00306=112823,838737,371446
BC00307=112823,838737,347276
BC00308=112823,838737,371446
BC00309=112823,838737,371446
BC00310=112823,838737,371446
BC00311=112823,838737,371446
BC00312=112823,838737,371446
BC00313=112823,838737,371446
BC00314=112823,838737,371446
BC00315=112823,838737,371446
BC00316=112823,838737,371446
BC00317=112823,842247,331141
BC00318=112823,838737,371446
BC00319=112823,838737,371446
BC00320=95917,841923,362982
BC00321=95917,841923,278580
BC00322=95918,841923,278577
BC00323=95918,841923,278577
BC00324=95918,841923,278577
BC00325=95918,841923,278577
BC00326=95918,841923,278580
BC00327=95917,841923,362982
BC00328=95917,841923,362982
BC00329=95917,841923,362982
BC00330=95917,841923,362982
BC00331=95917,841923,362982
BC00332=95917,841923,362982
BC00333=113760,802727,443486
BC00334=113760,802727,443486
BC00335=113760,802727,443486
BC00336=113760,802727,443486
BC00337=113760,802727,443486
BC00338=113760,802727,443486
BC00339=113760,802727,443486
BC00340=113760,802727,443486
BC00341=113760,802727,443486
BC00342=113760,802727,443486
BC00343=113760,802727,443486
BC00344=105225,809384,420294
BC00345=71151,822459,422634
BC00346=71151,822459,422634
BC00347=71151,822459,422634
BC00348=71151,822459,422634
BC00349=71151,822459,422634
BC00350=71151,822459,422634
BC00351=71151,822459,422634
BC00352=71151,822459,422634
BC00353=71151,822459,422634
BC00354=71151,822459,422634
BC00355=71151,822459,422634
BC00356=83716,796230,577321
BC00357=83716,796230,577321
BC00358=83716,796230,577321
BC00359=83716,796230,577321
BC00360=83716,796230,577321
BC00361=83716,796230,577321
BC00362=83716,796230,577321
BC00363=83716,796230,577321
BC00364=107468,821574,386040
BC00365=107468,821574,386040
BC00366=107468,821574,386040
BC00367=107468,821574,386040
BC00368=107468,821574,386040
BC00369=107468,821574,386040
BC00370=107468,821574,386040
BC00371=107468,821574,386040
BC00372=107468,821574,386040
BC00373=107468,821574,386040
BC00374=98517,821001,368440
BC00375=79840,837992,369859
BC00376=79840,837992,369859
BC00377=79840,837992,369859
BC00378=79840,837992,369859
BC00379=79840,837992,369859
BC00380=79840,837992,369859
BC00381=79840,837992,369859
BC00382=79840,837992,369859
BC00383=79840,837992,369859
BC00384=79840,837992,369859
BC00385=79840,837992,369859
BC00386=56247,787784,530537
BC00387=56247,787784,530537
BC00388=56247,787784,530537
BC00389=56247,787784,530537
BC00390=56247,787784,530537
BC00391=56247,787784,530537
BC00392=56247,787784,530537
BC00393=56247,787784,530537
BC00394=90098,809263,432129
BC00395=117602,826714,352172
BC00396=117602,826714,352172
BC00397=117602,826714,352172
BC00398=117602,826714,352172
BC00399=117602,826714,352172
BC00400=117602,826714,352172
BC00401=117602,826714,352172
BC00402=117602,826714,352172
BC00403=117602,826714,352172
BC00404=117602,826714,352172
BC00405=126877,832651,364221
BC00406=131515,835619,370246
BC00407=131515,835619,370246
BC00408=131515,835619,370246
BC00409=131515,835619,370246
BC00410=131515,835619,370246
BC00411=131515,835619,370246
BC00412=131515,835619,370246
BC00413=131515,835619,370246
BC00414=131515,835619,370246
BC00415=131515,835619,370246
BC00416=131515,835619,370246
BC00417=90780,809429,536518
BC00418=91468,810120,509844
BC00419=91743,810396,499175
BC00420=91743,810396,499175
BC00421=91743,810396,499175
BC00422=91745,811011,499181
BC00423=91470,810734,509851
BC00424=90782,810043,536525
BC00425=90780,809429,536518
BC00426=90780,677587,536518
BC00427=122178,711426,262582
BC00428=129566,724478,198127
BC00429=152481,738510,229723
BC00430=153188,743935,210842
BC00431=153471,746105,203290
BC00432=153471,746105,203290
BC00433=153471,746105,203290
BC00434=178419,747743,194040
BC00435=198738,754799,174592
BC00436=199704,755257,173467
BC00437=201481,753446,179748
BC00438=205924,748918,195450
BC00439=205914,748916,222334
BC00440=140861,743664,275053
BC00441=142200,745983,269639
BC00442=142200,745983,269639
BC00443=142200,745983,269639
BC00444=141326,745985,265401
BC00445=139461,745998,256423
BC00446=138579,746008,252202
BC00447=137239,743689,257616
BC00448=140861,743664,275053
BC00449=158142,738296,276224
BC00450=157676,736172,283618
BC00451=157686,736173,256734
BC00452=156866,741594,237889
BC00453=156538,743762,230351
BC00454=156538,743762,230351
BC00455=156538,743762,230351
BC00456=167187,744647,226440
BC00457=187251,751680,220156
BC00458=189813,752792,218066
BC00459=191590,750981,224347
BC00460=196033,746452,240049
BC00461=196012,746450,293816
BC00462=131888,717539,53
BC00463=131068,722959,53
BC00464=130740,725127,53
BC00465=130740,725127,53
BC00466=130740,725127,53
BC00467=139307,729508,53
BC00468=158758,734252,53
BC00469=161265,735929,53
BC00470=163042,734117,53
BC00471=167485,729589,53
BC00472=167464,729587,53
BC00473=109122,808327,293501
BC00474=110915,803765,284066
BC00475=110915,697318,284066
BC00476=308726,697318,147266
BC00477=398174,705389,4619
BC00478=398174,702811,16248
BC00479=398174,707203,53
BC00480=398174,705653,53
BC00481=398174,708960,53
BC00482=398174,708960,53
BC00483=398174,705653,53
BC00484=398174,705653,53
BC00485=398174,705653,53
BC00486=398174,705653,53
BC00487=398174,698596,1447
BC00488=398174,692515,17689
BC00489=264874,694777,10629
BC00490=251942,672671,69662
BC00491=174905,676397,197036
BC00492=246048,666220,100031
BC00493=249809,671543,85513
BC00494=251313,673683,79706
BC00495=251313,673683,79706
BC00496=251313,673683,79706
BC00497=250438,673684,75469
BC00498=248573,673697,66491
BC00499=247692,673708,62269
BC00500=246187,671568,68076
BC00501=242426,666217,82593
BC00502=199516,725910,40957
BC00503=203277,731261,26440
BC00504=204782,733401,20633
BC00505=204782,733401,20633
BC00506=204782,733401,20633
BC00507=203934,733402,16530
BC00508=202042,733415,7418
BC00509=201188,733426,3329
BC00510=199684,731286,9136
BC00511=195923,725935,23654
BC00512=195902,725933,77421
BC00513=197406,728073,71614
BC00514=197406,671867,269361
BC00515=197406,671867,269361
BC00516=156718,775147,252165
BC00517=132577,836422,356218
BC00518=132577,836422,204582
BC00519=132577,836422,241964
BC00520=132577,836422,241964
BC00521=132577,836422,241964
BC00522=132577,836422,241964
BC00523=132577,836422,241964
BC00524=132577,836422,241964
BC00525=132577,836422,222331
BC00526=132577,836422,186039
BC00527=117803,830955,65927
BC00528=113819,828411,65917
BC00529=106531,823737,65871
BC00530=106531,823737,65871
BC00531=106531,823737,65871
BC00532=106531,823737,65871
BC00533=106531,823737,65871
BC00534=111823,818035,92310
BC00535=155346,771391,566288
BC00536=197406,671867,536806
BC00537=197406,671867,269361
BC00538=259574,750536,237143
BC00539=311205,810481,212796
BC00540=311205,810481,212796
BC00541=311205,810481,212796
BC00542=311205,810481,212796
BC00543=311205,810481,212796
BC00544=311205,810481,212796
BC00545=311205,810481,212796
BC00546=311205,810481,212796
BC00547=311205,810481,212796
BC00548=311205,810481,212796
BC00549=311205,810481,212796
BC00550=311205,810481,212796
BC00551=311205,810481,212796
BC00552=311205,810481,212796
BC00553=311205,810481,212796
BC00554=311205,810481,212796
BC00555=311205,810481,212796
BC00556=311205,810481,212796
BC00557=311205,810481,212796
BC00558=311205,810481,212796
BC00559=311205,810481,212796
BC00560=311205,810481,212796
BC00561=311205,810481,212796
BC00562=311205,810481,212796
BC00563=311205,810481,212796
BC00564=311205,810481,212796
BC00565=311205,810481,212796
BC00566=311205,810481,212796
BC00567=311205,810481,212796
BC00568=311205,810481,212796
BC00569=311205,810481,212796
BC00570=311205,810481,212796
BC00571=311205,810481,212796
BC00572=311205,810481,212796
BC00573=311205,810481,212796
BC00574=311205,810481,212796
BC00575=311205,810481,212796
BC00576=311205,810481,212796
BC00577=311205,810481,212796
BC00578=311205,810481,212796
BC00579=311205,810481,212796
BC00580=311205,810481,212796
BC00581=311206,810481,212793
BC00582=311206,810481,212793
BC00583=311206,810481,212793
BC00584=311206,810481,212793
BC00585=311206,810481,212793
BC00586=311206,810481,212793
BC00587=311206,810481,212793
BC00588=311206,810481,212793
BC00589=315649,791685,239699
BC00590=344285,670537,413125
BC00591=148456,753848,427487
BC00592=149313,803884,512961
BC00593=149313,803884,314593
BC00594=149313,803884,267132
BC00595=149313,803884,314593
BC00596=149313,803884,314593
BC00597=149313,803884,314593
BC00598=149313,803884,314593
BC00599=149313,803884,314593
BC00600=149313,803884,314593
BC00601=149313,803884,314593
BC00602=149313,803884,314593
BC00603=199464,674570,1075173
EC00000=798156,1112951
EC00001=798156,1112951
EC00002=798156,1112951
EC00003=798156,1112951
EC00004=798156,1112951
EC00005=798156,1112951
EC00006=798156,1112951
EC00007=798156,1112951
EC00008=798156,1112951
EC00009=798156,1112951
EC00010=798156,1112951
EC00011=798156,1112951
EC00012=798156,1112951
EC00013=798156,1112951
EC00014=798156,1112951
EC00015=798156,1112951
EC00016=798156,1112951
EC00017=798156,1112951
EC00018=798156,1112951
EC00019=798156,1112951
EC00020=798156,1112951
EC00021=798156,1112951
EC00022=798156,1112951
EC00023=798156,1112951
EC00024=798155,1112950
EC00025=798156,1112951
EC00026=798156,1112951
EC00027=798156,1112951
EC00028=798156,1112951
EC00029=798156,1112951
EC00030=798156,1112951
EC00031=798156,1112951
EC00032=798156,1112951
EC00033=798156,1112951
EC00034=798156,1112951
EC00035=798156,1112951
EC00036=798156,1112951
EC00037=798156,1112951
EC00038=798156,1112951
EC00039=798156,1112951
EC00040=798156,1112951
EC00041=798156,1112951
EC00042=798156,1112951
EC00043=798156,1112951
EC00044=798156,1112951
EC00045=798156,1112951
EC00046=798156,1112951
EC00047=798156,1112951
EC00048=798156,1112951
EC00049=798156,1112951
EC00050=798156,1112951
EC00051=798156,1112951
EC00052=798156,1112951
EC00053=798156,1112951
EC00054=798156,1112951
EC00055=798156,1112951
EC00056=798156,1112951
EC00057=798156,1112951
EC00058=798156,1112951
EC00059=798156,1112951
EC00060=798156,1112951
EC00061=798156,1112951
EC00062=798156,1112951
EC00063=798156,1112951
EC00064=798156,1112951
EC00065=798156,1112951
EC00066=798156,1112951
EC00067=798156,1112951
EC00068=798156,1112951
EC00069=798156,1112951
EC00070=798156,1112951
EC00071=798156,1112951
EC00072=798155,1112950
EC00073=798155,1112950
EC00074=798155,1112950
EC00075=798155,1112950
EC00076=798155,1112950
EC00077=798155,1112950
EC00078=798155,1112950
EC00079=798155,1112950
EC00080=798155,1112950
EC00081=798155,1112950
EC00082=798155,1112950
EC00083=798154,1112950
EC00084=798154,1112950
EC00085=798154,1112950
EC00086=798154,1112950
EC00087=798154,1112950
EC00088=798154,1112950
EC00089=798154,1112950
EC00090=798152,1112948
EC00091=798152,1112948
EC00092=798152,1112948
EC00093=798152,1112948
EC00094=798152,1112948
EC00095=798152,1112948
EC00096=798152,1112948
EC00097=798152,1112948
EC00098=798152,1112948
EC00099=798152,1112948
EC00100=798152,1112948
EC00101=798152,1112948
EC00102=798152,1112948
EC00103=798152,1112948
EC00104=798152,1112948
EC00105=798152,1112948
EC00106=798152,1112948
EC00107=798152,1112948
EC00108=798152,1112948
EC00109=798152,1112948
EC00110=798152,1112948
EC00111=798152,1112948
EC00112=798152,1112948
EC00113=798152,1112948
EC00114=798152,1112948
EC00115=798152,1112948
EC00116=798152,1112948
EC00117=798152,1112948
EC00118=798152,1112948
EC00119=798152,1112948
EC00120=798152,1112948
EC00121=798152,1112948
EC00122=798152,1112948
EC00123=798152,1112948
EC00124=798152,1112948
EC00125=798152,1112948
EC00126=798152,1112948
EC00127=798152,1112948
EC00128=798152,1112948
EC00129=798152,1112948
EC00130=798152,1112948
EC00131=798152,1112948
EC00132=798152,1112948
EC00133=798152,1112948
EC00134=798156,1112951
EC00135=910680,1112951
EC00136=953239,1112951
EC00137=960687,1112951
EC00138=975524,1112951
EC00139=975524,1112951
EC00140=975524,1112951
EC00141=975524,1112951
EC00142=975524,1112951
EC00143=975524,1112951
EC00144=975524,1112951
EC00145=975524,1112951
EC00146=975524,1112951
EC00147=975524,1112951
EC00148=975524,1112951
EC00149=975524,1112951
EC00150=975524,1112951
EC00151=975524,1112951
EC00152=975524,1112951
EC00153=975524,1112951
EC00154=975524,1112951
EC00155=975524,1112951
EC00156=975524,1112951
EC00157=975524,1112951
EC00158=975524,1112951
EC00159=975524,1112951
EC00160=975524,1112951
EC00161=975524,1112951
EC00162=975524,1112951
EC00163=975524,1112951
EC00164=975524,1112951
EC00165=975521,1112950
EC00166=975524,1112951
EC00167=975524,1112951
EC00168=975524,1112951
EC00169=975524,1112951
EC00170=975524,1112951
EC00171=975524,1112951
EC00172=975524,1112951
EC00173=975524,1112951
EC00174=975524,1112951
EC00175=975524,1112951
EC00176=975524,1112951
EC00177=975524,1112951
EC00178=975524,1112951
EC00179=975524,1112951
EC00180=975524,1112951
EC00181=975524,1112951
EC00182=975524,1112951
EC00183=975524,1112951
EC00184=975524,1112951
EC00185=975524,1112951
EC00186=975524,1112951
EC00187=975524,1112951
EC00188=975524,1112951
EC00189=975524,1112951
EC00190=975524,1112951
EC00191=975524,1112951
EC00192=975524,1112951
EC00193=975524,1112951
EC00194=975524,1112951
EC00195=975521,1112951
EC00196=975524,1112951
EC00197=975524,1112951
EC00198=975521,1112951
EC00199=975521,1112951
EC00200=975521,1112951
EC00201=975521,1112951
EC00202=975524,1112951
EC00203=975524,1112951
EC00204=975524,1112951
EC00205=975524,1112951
EC00206=975524,1112951
EC00207=975524,1112951
EC00208=975524,1112951
EC00209=975524,1112951
EC00210=975524,1112951
EC00211=975524,1112951
EC00212=975524,1112951
EC00213=975524,1112951
EC00214=975524,1112951
EC00215=975524,1112951
EC00216=975524,1112951
EC00217=975524,1112951
EC00218=975524,1112951
EC00219=975524,1112951
EC00220=975524,1112951
EC00221=975524,1112951
EC00222=975524,1112951
EC00223=975524,1112951
EC00224=975524,1112951
EC00225=975524,1112951
EC00226=975524,1112951
EC00227=975524,1112951
EC00228=975524,1112951
EC00229=975524,1112951
EC00230=975524,1112951
EC00231=975524,1112951
EC00232=975524,1112951
EC00233=975524,1112951
EC00234=975524,1112951
EC00235=975524,1112951
EC00236=975524,1112951
EC00237=975524,1112951
EC00238=975524,1112951
EC00239=975524,1112951
EC00240=975524,1112951
EC00241=975524,1112951
EC00242=975524,1112951
EC00243=975524,1112951
EC00244=975524,1112951
EC00245=975524,1112951
EC00246=975524,1112951
EC00247=975524,1112951
EC00248=975524,1112951
EC00249=975524,1112951
EC00250=975524,1112951
EC00251=975524,1112951
EC00252=975524,1112951
EC00253=975524,1112951
EC00254=975524,1112951
EC00255=975524,1112951
EC00256=975524,1112951
EC00257=975524,1112951
EC00258=975524,1112951
EC00259=975524,1112951
EC00260=975524,1112951
EC00261=975524,1112951
EC00262=975512,1112947
EC00263=975524,1112951
EC00264=975524,1112951
EC00265=975515,1112948
EC00266=975524,1112951
EC00267=975524,1112951
EC00268=975521,1112950
EC00269=975524,1112951
EC00270=975524,1112951
EC00271=975524,1112951
EC00272=975524,1112951
EC00273=975524,1112951
EC00274=975524,1112951
EC00275=975524,1112951
EC00276=975524,1112951
EC00277=975524,1112951
EC00278=975524,1112951
EC00279=975524,1112951
EC00280=975524,1112951
EC00281=975524,1112951
EC00282=975524,1112951
EC00283=975524,1112951
EC00284=975524,1112951
EC00285=975524,1112951
EC00286=975524,1112951
EC00287=975524,1112951
EC00288=975524,1112951
EC00289=975524,1112951
EC00290=798156,1112951
EC00291=798156,1112951
EC00292=798156,1112951
EC00293=798156,1112951
EC00294=798156,1112951
EC00295=798156,1112951
EC00296=798156,1112951
EC00297=798156,1112951
EC00298=798156,1112951
EC00299=798156,1112951
EC00300=798156,1112951
EC00301=798156,1112951
EC00302=798156,1112951
EC00303=798156,1112951
EC00304=798156,1112951
EC00305=798156,1112951
EC00306=798156,1112951
EC00307=798156,1112951
EC00308=798156,1112951
EC00309=798156,1112951
EC00310=798156,1112951
EC00311=798156,1112951
EC00312=798156,1112951
EC00313=798156,1112951
EC00314=798156,1112951
EC00315=798156,1112951
EC00316=798156,1112951
EC00317=798155,1112950
EC00318=798156,1112951
EC00319=798156,1112951
EC00320=798156,1112951
EC00321=798156,1112951
EC00322=798155,1112950
EC00323=798155,1112950
EC00324=798155,1112950
EC00325=798155,1112950
EC00326=798155,1112950
EC00327=798156,1112951
EC00328=798156,1112951
EC00329=798156,1112951
EC00330=798156,1112951
EC00331=798156,1112951
EC00332=798156,1112951
EC00333=798156,1112951
EC00334=798156,1112951
EC00335=798156,1112951
EC00336=798156,1112951
EC00337=798156,1112951
EC00338=798156,1112951
EC00339=798156,1112951
EC00340=798156,1112951
EC00341=798156,1112951
EC00342=798156,1112951
EC00343=798156,1112951
EC00344=798156,1112951
EC00345=798156,1112951
EC00346=798156,1112951
EC00347=798156,1112951
EC00348=798156,1112951
EC00349=798156,1112951
EC00350=798156,1112951
EC00351=798156,1112951
EC00352=798156,1112951
EC00353=798156,1112951
EC00354=798156,1112951
EC00355=798156,1112951
EC00356=798156,1112951
EC00357=798156,1112951
EC00358=798156,1112951
EC00359=798156,1112951
EC00360=798156,1112951
EC00361=798156,1112951
EC00362=798156,1112951
EC00363=798156,1112951
EC00364=798156,1112951
EC00365=798156,1112951
EC00366=798156,1112951
EC00367=798156,1112951
EC00368=798156,1112951
EC00369=798156,1112951
EC00370=798156,1112951
EC00371=798156,1112951
EC00372=798156,1112951
EC00373=798156,1112951
EC00374=798156,1112951
EC00375=798156,1112951
EC00376=798156,1112951
EC00377=798156,1112951
EC00378=798156,1112951
EC00379=798156,1112951
EC00380=798156,1112951
EC00381=798156,1112951
EC00382=798156,1112951
EC00383=798156,1112951
EC00384=798156,1112951
EC00385=798156,1112951
EC00386=798156,1112951
EC00387=798156,1112951
EC00388=798156,1112951
EC00389=798156,1112951
EC00390=798156,1112951
EC00391=798156,1112951
EC00392=798156,1112951
EC00393=798156,1112951
EC00394=798156,1112951
EC00395=798156,1112951
EC00396=798156,1112951
EC00397=798156,1112951
EC00398=798156,1112951
EC00399=798156,1112951
EC00400=798156,1112951
EC00401=798156,1112951
EC00402=798156,1112951
EC00403=798156,1112951
EC00404=798156,1112951
EC00405=798156,1112951
EC00406=798156,1112951
EC00407=798156,1112951
EC00408=798156,1112951
EC00409=798156,1112951
EC00410=798156,1112951
EC00411=798156,1112951
EC00412=798156,1112951
EC00413=798156,1112951
EC00414=798156,1112951
EC00415=798156,1112951
EC00416=798156,1112951
EC00417=798156,1112951
EC00418=798156,1112951
EC00419=798156,1112951
EC00420=798156,1112951
EC00421=798156,1112951
EC00422=798156,1112951
EC00423=798156,1112951
EC00424=798156,1112951
EC00425=798156,1112951
EC00426=798156,1112951
EC00427=798156,1112951
EC00428=798156,1112951
EC00429=798156,1112951
EC00430=798156,1112951
EC00431=798156,1112951
EC00432=798156,1112951
EC00433=798156,1112951
EC00434=798156,1112951
EC00435=798156,1112951
EC00436=798156,1112951
EC00437=798156,1112951
EC00438=798156,1112951
EC00439=798156,1112951
EC00440=798156,1112951
EC00441=798156,1112951
EC00442=798156,1112951
EC00443=798156,1112951
EC00444=798156,1112951
EC00445=798156,1112951
EC00446=798156,1112951
EC00447=798156,1112951
EC00448=798156,1112951
EC00449=798156,1112951
EC00450=798156,1112951
EC00451=798156,1112951
EC00452=798156,1112951
EC00453=798156,1112951
EC00454=798156,1112951
EC00455=798156,1112951
EC00456=798156,1112951
EC00457=798156,1112951
EC00458=798156,1112951
EC00459=798156,1112951
EC00460=798156,1112951
EC00461=798156,1112951
EC00462=798156,1112951
EC00463=798156,1112951
EC00464=798156,1112951
EC00465=798156,1112951
EC00466=798156,1112951
EC00467=798156,1112951
EC00468=798156,1112951
EC00469=798156,1112951
EC00470=798156,1112951
EC00471=798156,1112951
EC00472=798156,1112951
EC00473=798156,1112951
EC00474=798156,1112951
EC00475=798156,1112951
EC00476=798156,1112951
EC00477=798156,1112951
EC00478=798156,1112951
EC00479=798156,1112951
EC00480=798156,1112951
EC00481=798156,1112951
EC00482=798156,1112951
EC00483=798156,1112951
EC00484=798156,1112951
EC00485=798156,1112951
EC00486=798156,1112951
EC00487=798156,1112951
EC00488=798156,1112951
EC00489=798156,1112951
EC00490=798156,1112951
EC00491=798156,1112951
EC00492=798156,1112951
EC00493=798156,1112951
EC00494=798156,1112951
EC00495=798156,1112951
EC00496=798156,1112951
EC00497=798156,1112951
EC00498=798156,1112951
EC00499=798156,1112951
EC00500=798156,1112951
EC00501=798156,1112951
EC00502=798156,1112951
EC00503=798156,1112951
EC00504=798156,1112951
EC00505=798156,1112951
EC00506=798156,1112951
EC00507=798156,1112951
EC00508=798156,1112951
EC00509=798156,1112951
EC00510=798156,1112951
EC00511=798156,1112951
EC00512=798156,1112951
EC00513=798156,1112951
EC00514=798156,1112951
EC00515=798156,1112951
EC00516=798155,1112951
EC00517=798156,1112951
EC00518=798156,1112951
EC00519=798156,1112951
EC00520=798156,1112951
EC00521=798156,1112951
EC00522=798156,1112951
EC00523=798156,1112951
EC00524=798156,1112951
EC00525=798156,1112951
EC00526=798156,1112951
EC00527=798156,1112951
EC00528=798156,1112951
EC00529=798156,1112951
EC00530=798156,1112951
EC00531=798156,1112951
EC00532=798156,1112951
EC00533=798156,1112951
EC00534=798156,1112951
EC00535=798156,1112951
EC00536=798156,1112951
EC00537=798156,1112951
EC00538=798156,1112951
EC00539=798156,1112951
EC00540=798156,1112951
EC00541=798156,1112951
EC00542=798156,1112951
EC00543=798156,1112951
EC00544=798156,1112951
EC00545=798156,1112951
EC00546=798156,1112951
EC00547=798156,1112951
EC00548=798156,1112951
EC00549=798156,1112951
EC00550=798156,1112951
EC00551=798156,1112951
EC00552=798156,1112951
EC00553=798156,1112951
EC00554=798156,1112951
EC00555=798156,1112951
EC00556=798156,1112951
EC00557=798156,1112951
EC00558=798156,1112951
EC00559=798156,1112951
EC00560=798156,1112951
EC00561=798156,1112951
EC00562=798156,1112951
EC00563=798156,1112951
EC00564=798156,1112951
EC00565=798156,1112951
EC00566=798156,1112951
EC00567=798156,1112951
EC00568=798156,1112951
EC00569=798156,1112951
EC00570=798156,1112951
EC00571=798156,1112951
EC00572=798156,1112951
EC00573=798156,1112951
EC00574=798156,1112951
EC00575=798156,1112951
EC00576=798156,1112951
EC00577=798156,1112951
EC00578=798156,1112951
EC00579=798156,1112951
EC00580=798156,1112951
EC00581=798155,1112950
EC00582=798155,1112950
EC00583=798155,1112950
EC00584=798155,1112950
EC00585=798155,1112950
EC00586=798155,1112950
EC00587=798155,1112950
EC00588=798155,1112950
EC00589=798155,1112950
EC00590=798156,1112951
EC00591=798156,1112951
EC00592=798156,1112951
EC00593=798156,1112951
EC00594=798156,1112951
EC00595=798156,1112951
EC00596=798156,1112951
EC00597=798156,1112951
EC00598=798156,1112951
EC00599=798156,1112951
EC00600=798156,1112951
EC00601=798156,1112951
EC00602=798156,1112951
EC00603=798155,1112950
///POSTYPE BASE
///RECTAN
///RCONF 0,0,0,0,0,0,0,0,0,0,0,0,0,0,0,0,0,0,0,0,0,0,0,0
P00006=0.222,-3.123,-1.508,0.0000,0.0000,0.0000
P00021=-0.225,-6.128,-0.405,0.0000,0.0000,0.0000
P00022=0.222,-3.123,-1.508,0.0000,0.0000,0.0000
P00023=0.143,-0.036,0.682,0.0000,0.0000,0.0000
P00024=0.145,-0.552,1.326,0.0000,0.0000,0.0000
P00025=-2.003,0.006,0.728,0.0000,0.0000,0.0000
P00026=0.562,-0.002,-0.337,0.0000,0.0000,0.0000
P00027=-0.746,0.015,-9.096,0.0000,0.0000,0.0000
P00031=1.853,-0.001,-1.549,0.0000,0.0000,0.0000
P00032=1.957,0.503,-7.217,0.0000,0.0000,0.0000
///RCONF 0,0,0,0,1,0,0,0,0,0,0,0,0,0,0,0,0,0,0,0,0,0,0,0
P00033=-0.123,0.612,-5.012,0.0000,0.0000,0.0000
///RCONF 0,0,0,0,0,0,0,0,0,0,0,0,0,0,0,0,0,0,0,0,0,0,0,0
P00034=-0.304,0.773,-2.693,0.0000,0.0000,0.0000
P00035=2.817,0.591,-1.622,0.0000,0.0000,0.0000
P00036=-1.108,-0.829,1.850,0.0000,0.0000,0.0000
P00041=0.192,3.924,0.305,0.0000,0.0000,0.0000
P00042=-0.217,1.941,0.413,0.0000,0.0000,0.0000
P00043=-0.044,-1.937,1.197,0.0000,0.0000,0.0000
P00044=0.687,-2.322,1.156,0.0000,0.0000,0.0000
P00045=-0.068,-0.810,1.603,0.0000,0.0000,0.0000
P00046=0.799,0.043,1.292,0.0000,0.0000,0.0000
P00088=-2.376,0.094,2.453,0.0000,0.0000,0.0000
P00089=5.697,-3.100,-1.263,0.0000,0.0000,0.0000
P00090=0.184,3.539,2.293,0.0000,0.0000,0.0000
//INST
///DATE 2025/01/29 13:52
///ATTR SC,RW
///GROUP1 RB1,BS1
///GROUP2 ST1
NOP
'OK_r2_O57-69(2)(90,0)2
'Down
SFTOF3D
MOVJ C00000 BC00000 VJ=100.00  +MOVJ EC00000 VJ=100.00
MOVL C00001 BC00001 V=400.0  +MOVJ EC00001 VJ=100.00
SMOVL C00002 BC00002 V=166.7  +MOVJ EC00002
SREFP 3 C00003 BC00003  +REFP EC00003
CALL JOB:SEARCH-R1-S13D
SET P026 P006
SFTON3D P026
SMOVL C00004 BC00004 V=166.7  +MOVJ EC00004
SREFP 3 C00005 BC00005  +REFP EC00005
CALL JOB:SEARCH-R1-S13D
SET P026 P006
SFTON3D P026
SMOVL C00006 BC00006 V=166.7  +MOVJ EC00006
MOVL C00007 BC00007 V=400.0  +MOVJ EC00007 VJ=100.00
MOVL C00008 BC00008 V=1000.0  +MOVJ EC00008 VJ=100.00
'Path S3529
SFTOF3D
MOVJ C00009 BC00009 VJ=100.00  +MOVJ EC00009 VJ=100.00
MOVL C00010 BC00010 V=400.0  +MOVJ EC00010 VJ=100.00
SMOVL C00011 BC00011 V=166.7  +MOVJ EC00011
SREFP 3 C00012 BC00012  +REFP EC00012
CALL JOB:SEARCH-R1-S13D
SET P027 P006
SFTON3D P027
SMOVL C00013 BC00013 V=166.7  +MOVJ EC00013
SREFP 3 C00014 BC00014  +REFP EC00014
CALL JOB:SEARCH-R1-S13D
SET P027 P006
SFTON3D P027
SMOVL C00015 BC00015 V=166.7  +MOVJ EC00015
MOVL C00016 BC00016 V=400.0  +MOVJ EC00016 VJ=100.00
MOVL C00017 BC00017 V=1000.0  +MOVJ EC00017 VJ=100.00
MOVL C00018 BC00018 V=1000.0  +MOVJ EC00018 VJ=100.00
'Path S3530
SFTOF3D
MOVJ C00019 BC00019 VJ=100.00  +MOVJ EC00019 VJ=100.00
COMM PAUSE
COMM MOVL C00020 BC00020 V=400.0  +MOVJ EC00020 VJ=100.00
COMM SMOVL C00021 BC00021 V=166.7  +MOVJ EC00021
COMM SREFP 3 C00022 BC00022  +REFP EC00022
COMM CALL JOB:SEARCH-R1-S13D
COMM SET P022 P006
COMM SFTON3D P022
COMM SMOVL C00023 BC00023 V=166.7  +MOVJ EC00023
COMM SREFP 3 C00024 BC00024  +REFP EC00024
COMM CALL JOB:SEARCH-R1-S13D
COMM SET P022 P006
COMM SFTON3D P022
COMM SMOVL C00025 BC00025 V=166.7  +MOVJ EC00025
SFTOF3D
MOVL C00026 BC00026 V=1000.0  +MOVJ EC00026 VJ=100.00
SMOVL C00027 BC00027 V=1000.0  +MOVJ EC00027
SMOVL C00028 BC00028 V=166.7  +MOVJ EC00028
SREFP 3 C00029 BC00029  +REFP EC00029
CALL JOB:SEARCH-R1-S13D
SET P088 P006
SFTON3D P088
SMOVL C00030 BC00030 V=166.7  +MOVJ EC00030
SMOVL C00031 BC00031 V=166.7  +MOVJ EC00031
SMOVL C00032 BC00032 V=166.7  +MOVJ EC00032
SREFP 3 C00033 BC00033  +REFP EC00033
CALL JOB:SEARCH-R1-S13D
SET P088 P006
SFTON3D P088
SMOVL C00034 BC00034 V=166.7  +MOVJ EC00034
SFTOF3D
SMOVL C00035 BC00035 V=1000.0  +MOVJ EC00035
MOVJ C00036 BC00036 VJ=100.00  +MOVJ EC00036 VJ=100.00
MOVJ C00037 BC00037 VJ=100.00  +MOVJ EC00037 VJ=100.00
MOVL C00038 BC00038 V=400.0  +MOVJ EC00038 VJ=100.00
SMOVL C00039 BC00039 V=133.3  +MOVJ EC00039
SREFP 3 C00040 BC00040  +REFP EC00040
CALL JOB:SEARCH-R1-S13D
SET P021 P006
SFTON3D P021
SMOVL C00041 BC00041 V=166.7  +MOVJ EC00041
SREFP 3 C00042 BC00042  +REFP EC00042
CALL JOB:SEARCH-R1-S13D
SET P021 P006
SFTON3D P021
SMOVL C00043 BC00043 V=166.7  +MOVJ EC00043
SMOVL C00044 BC00044 V=166.7  +MOVJ EC00044
SREFP 3 C00045 BC00045  +REFP EC00045
CALL JOB:SEARCH-R1-S13D
SET P021 P006
SFTON3D P021
SMOVL C00046 BC00046 V=166.7  +MOVJ EC00046
MOVL C00047 BC00047 V=400.0  +MOVJ EC00047 VJ=100.00
MOVL C00048 BC00048 V=1000.0  +MOVJ EC00048 VJ=100.00
MOVJ C00049 BC00049 VJ=100.00  +MOVJ EC00049 VJ=100.00
MOVJ C00050 BC00050 VJ=100.00  +MOVJ EC00050 VJ=100.00
'Path S3538
SFTOF3D
MOVJ C00051 BC00051 VJ=100.00  +MOVJ EC00051 VJ=100.00
MOVL C00052 BC00052 V=400.0  +MOVJ EC00052 VJ=100.00
SMOVL C00053 BC00053 V=166.7  +MOVJ EC00053
SREFP 3 C00054 BC00054  +REFP EC00054
CALL JOB:SEARCH-R1-S13D
SET P032 P006
SFTON3D P032
SMOVL C00055 BC00055 V=166.7  +MOVJ EC00055
SREFP 3 C00056 BC00056  +REFP EC00056
CALL JOB:SEARCH-R1-S13D
SET P032 P006
SFTON3D P032
SMOVL C00057 BC00057 V=166.7  +MOVJ EC00057
SFTOF3D
MOVL C00058 BC00058 V=400.0  +MOVJ EC00058 VJ=100.00
MOVL C00059 BC00059 V=1000.0  +MOVJ EC00059 VJ=100.00
MOVJ C00060 BC00060 VJ=100.00  +MOVJ EC00060 VJ=100.00
MOVJ C00061 BC00061 VJ=100.00  +MOVJ EC00061 VJ=100.00
COMM PAUSE
COMM MOVJ C00062 BC00062 VJ=100.00  +MOVJ EC00062 VJ=100.00
COMM SMOVL C00063 BC00063 V=1000.0  +MOVJ EC00063
COMM SMOVL C00064 BC00064 V=166.7  +MOVJ EC00064
COMM SREFP 3 C00065 BC00065  +REFP EC00065
COMM CALL JOB:SEARCH-R1-S13D
COMM SET P089 P006
COMM SFTON3D P089
COMM SMOVL C00066 BC00066 V=166.7  +MOVJ EC00066
COMM SMOVL C00067 BC00067 V=166.7  +MOVJ EC00067
COMM SMOVL C00068 BC00068 V=166.7  +MOVJ EC00068
COMM SREFP 3 C00069 BC00069  +REFP EC00069
COMM CALL JOB:SEARCH-R1-S13D
COMM SET P089 P006
COMM SFTON3D P089
COMM SMOVL C00070 BC00070 V=166.7  +MOVJ EC00070
COMM SFTOF3D
SMOVL C00071 BC00071 V=1000.0  +MOVJ EC00071
SMOVL C00072 BC00072 V=1000.0  +MOVJ EC00072
SMOVL C00073 BC00073 V=166.7  +MOVJ EC00073
SREFP 3 C00074 BC00074  +REFP EC00074
CALL JOB:SEARCH-R1-S13D
SET P090 P006
SFTON3D P090
SMOVL C00075 BC00075 V=166.7  +MOVJ EC00075
SREFP 3 C00076 BC00076  +REFP EC00076
CALL JOB:SEARCH-R1-S13D
SET P090 P006
SFTON3D P090
SMOVL C00077 BC00077 V=166.7  +MOVJ EC00077
SMOVL C00078 BC00078 V=166.7  +MOVJ EC00078
SREFP 3 C00079 BC00079  +REFP EC00079
CALL JOB:SEARCH-R1-S13D
SET P090 P006
SFTON3D P090
SMOVL C00080 BC00080 V=250.0  +MOVJ EC00080
SFTOF3D
SMOVL C00081 BC00081 V=1000.0  +MOVJ EC00081
SMOVL C00082 BC00082 V=1000.0  +MOVJ EC00082
SMOVL C00083 BC00083 V=166.7  +MOVJ EC00083
SREFP 3 C00084 BC00084  +REFP EC00084
CALL JOB:SEARCH-R1-S13D
SET P031 P006
SFTON3D P031
SMOVL C00085 BC00085 V=166.7  +MOVJ EC00085
SMOVL C00086 BC00086 V=166.7  +MOVJ EC00086
SMOVL C00087 BC00087 V=166.7  +MOVJ EC00087
SREFP 3 C00088 BC00088  +REFP EC00088
CALL JOB:SEARCH-R1-S13D
SET P031 P006
SFTON3D P031
SMOVL C00089 BC00089 V=166.7  +MOVJ EC00089
SMOVL C00090 BC00090 V=166.7  +MOVJ EC00090
SMOVL C00091 BC00091 V=166.7  +MOVJ EC00091
SREFP 3 C00092 BC00092  +REFP EC00092
CALL JOB:SEARCH-R1-S13D
SET P031 P006
SFTON3D P031
SMOVL C00093 BC00093 V=166.7  +MOVJ EC00093
SMOVL C00094 BC00094 V=666.7  +MOVJ EC00094
SREFP 3 C00095 BC00095  +REFP EC00095
CALL JOB:SEARCH-R1-S13D
SET P032 P006
SFTON3D P032
SMOVL C00096 BC00096 V=166.7  +MOVJ EC00096
SMOVL C00097 BC00097 V=166.7  +MOVJ EC00097
SMOVL C00098 BC00098 V=166.7  +MOVJ EC00098
SREFP 3 C00099 BC00099  +REFP EC00099
CALL JOB:SEARCH-R1-S13D
SET P032 P006
SFTON3D P032
SMOVL C00100 BC00100 V=166.7  +MOVJ EC00100
SMOVL C00101 BC00101 V=666.7  +MOVJ EC00101
SMOVL C00102 BC00102 V=666.7  +MOVJ EC00102
SMOVL C00103 BC00103 V=166.7  +MOVJ EC00103
SREFP 3 C00104 BC00104  +REFP EC00104
CALL JOB:SEARCH-R1-S13D
SET P033 P006
SFTON3D P033
SMOVL C00105 BC00105 V=166.7  +MOVJ EC00105
SMOVL C00106 BC00106 V=166.7  +MOVJ EC00106
SMOVL C00107 BC00107 V=166.7  +MOVJ EC00107
SREFP 3 C00108 BC00108  +REFP EC00108
CALL JOB:SEARCH-R1-S13D
SET P033 P006
SFTON3D P033
SMOVL C00109 BC00109 V=166.7  +MOVJ EC00109
SMOVL C00110 BC00110 V=666.7  +MOVJ EC00110
SMOVL C00111 BC00111 V=166.7  +MOVJ EC00111
SREFP 3 C00112 BC00112  +REFP EC00112
CALL JOB:SEARCH-R1-S13D
SET P034 P006
SFTON3D P034
SMOVL C00113 BC00113 V=166.7  +MOVJ EC00113
SMOVL C00114 BC00114 V=166.7  +MOVJ EC00114
SMOVL C00115 BC00115 V=166.7  +MOVJ EC00115
SREFP 3 C00116 BC00116  +REFP EC00116
CALL JOB:SEARCH-R1-S13D
SET P034 P006
SFTON3D P034
SMOVL C00117 BC00117 V=166.7  +MOVJ EC00117
SMOVL C00118 BC00118 V=666.7  +MOVJ EC00118
SMOVL C00119 BC00119 V=166.7  +MOVJ EC00119
SREFP 3 C00120 BC00120  +REFP EC00120
CALL JOB:SEARCH-R1-S13D
SET P035 P006
SFTON3D P035
SMOVL C00121 BC00121 V=166.7  +MOVJ EC00121
SMOVL C00122 BC00122 V=166.7  +MOVJ EC00122
SMOVL C00123 BC00123 V=166.7  +MOVJ EC00123
SREFP 3 C00124 BC00124  +REFP EC00124
CALL JOB:SEARCH-R1-S13D
SET P035 P006
SFTON3D P035
SMOVL C00125 BC00125 V=166.7  +MOVJ EC00125
SMOVL C00126 BC00126 V=666.7  +MOVJ EC00126
SMOVL C00127 BC00127 V=166.7  +MOVJ EC00127
SREFP 3 C00128 BC00128  +REFP EC00128
CALL JOB:SEARCH-R1-S13D
SET P036 P006
SFTON3D P036
SMOVL C00129 BC00129 V=166.7  +MOVJ EC00129
SMOVL C00130 BC00130 V=166.7  +MOVJ EC00130
SMOVL C00131 BC00131 V=166.7  +MOVJ EC00131
SREFP 3 C00132 BC00132  +REFP EC00132
CALL JOB:SEARCH-R1-S13D
SET P036 P006
SFTON3D P036
SMOVL C00133 BC00133 V=166.7  +MOVJ EC00133
SFTOF3D
SMOVL C00134 BC00134 V=1000.0  +MOVJ EC00134
MOVJ C00135 BC00135 VJ=100.00  +MOVJ EC00135 VJ=100.00
'Up
MOVJ C00136 BC00136 VJ=100.00  +MOVJ EC00136 VJ=100.00
MOVJ C00137 BC00137 VJ=100.00  +MOVJ EC00137 VJ=100.00
'Path S3539
SFTOF3D
MOVJ C00138 BC00138 VJ=100.00  +MOVJ EC00138 VJ=100.00
MOVL C00139 BC00139 V=400.0  +MOVJ EC00139 VJ=100.00
SMOVL C00140 BC00140 V=100.0  +MOVJ EC00140
SREFP 3 C00141 BC00141  +REFP EC00141
CALL JOB:SEARCH-R1-S13D
SET P046 P006
SFTON3D P046
SMOVL C00142 BC00142 V=100.0  +MOVJ EC00142
SREFP 3 C00143 BC00143  +REFP EC00143
CALL JOB:SEARCH-R1-S13D
SET P046 P006
SFTON3D P046
SMOVL C00144 BC00144 V=100.0  +MOVJ EC00144
MOVL C00145 BC00145 V=400.0  +MOVJ EC00145 VJ=100.00
MOVL C00146 BC00146 V=1000.0  +MOVJ EC00146 VJ=100.00
'Path S3540
SFTOF3D
MOVJ C00147 BC00147 VJ=100.00  +MOVJ EC00147 VJ=100.00
MOVL C00148 BC00148 V=400.0  +MOVJ EC00148 VJ=100.00
SMOVL C00149 BC00149 V=100.0  +MOVJ EC00149
SREFP 3 C00150 BC00150  +REFP EC00150
CALL JOB:SEARCH-R1-S13D
SET P045 P006
SFTON3D P045
SMOVL C00151 BC00151 V=100.0  +MOVJ EC00151
SREFP 3 C00152 BC00152  +REFP EC00152
CALL JOB:SEARCH-R1-S13D
SET P045 P006
SFTON3D P045
SMOVL C00153 BC00153 V=100.0  +MOVJ EC00153
SREFP 3 C00154 BC00154  +REFP EC00154
CALL JOB:SEARCH-R1-S13D
SET P045 P006
SFTON3D P045
SMOVL C00155 BC00155 V=100.0  +MOVJ EC00155
MOVL C00156 BC00156 V=400.0  +MOVJ EC00156 VJ=100.00
MOVL C00157 BC00157 V=1000.0  +MOVJ EC00157 VJ=100.00
MOVL C00158 BC00158 V=1000.0  +MOVJ EC00158 VJ=100.00
MOVJ C00159 BC00159 VJ=100.00  +MOVJ EC00159 VJ=50.00
SFTOF3D
MOVJ C00160 BC00160 VJ=100.00  +MOVJ EC00160 VJ=50.00
MOVJ C00161 BC00161 VJ=100.00  +MOVJ EC00161 VJ=100.00
MOVL C00162 BC00162 V=400.0  +MOVJ EC00162 VJ=100.00
SMOVL C00163 BC00163 V=100.0  +MOVJ EC00163
SREFP 3 C00164 BC00164  +REFP EC00164
CALL JOB:SEARCH-R1-S13D
SET P043 P006
SFTON3D P043
SMOVL C00165 BC00165 V=100.0  +MOVJ EC00165
SREFP 3 C00166 BC00166  +REFP EC00166
CALL JOB:SEARCH-R1-S13D
SET P043 P006
SFTON3D P043
SMOVL C00167 BC00167 V=100.0  +MOVJ EC00167
SREFP 3 C00168 BC00168  +REFP EC00168
CALL JOB:SEARCH-R1-S13D
SET P043 P006
SFTON3D P043
SMOVL C00169 BC00169 V=100.0  +MOVJ EC00169
MOVL C00170 BC00170 V=400.0  +MOVJ EC00170 VJ=100.00
MOVL C00171 BC00171 V=1000.0  +MOVJ EC00171 VJ=100.00
'Path S3543
SFTOF3D
MOVJ C00172 BC00172 VJ=100.00  +MOVJ EC00172 VJ=100.00
MOVL C00173 BC00173 V=400.0  +MOVJ EC00173 VJ=100.00
SMOVL C00174 BC00174 V=100.0  +MOVJ EC00174
SREFP 3 C00175 BC00175  +REFP EC00175
CALL JOB:SEARCH-R1-S13D
SET P042 P006
SFTON3D P042
SMOVL C00176 BC00176 V=100.0  +MOVJ EC00176
SREFP 3 C00177 BC00177  +REFP EC00177
CALL JOB:SEARCH-R1-S13D
SET P042 P006
SFTON3D P042
SMOVL C00178 BC00178 V=100.0  +MOVJ EC00178
SREFP 3 C00179 BC00179  +REFP EC00179
CALL JOB:SEARCH-R1-S13D
SET P042 P006
SFTON3D P042
SMOVL C00180 BC00180 V=100.0  +MOVJ EC00180
MOVL C00181 BC00181 V=1000.0  +MOVJ EC00181 VJ=100.00
'Path S3544
SFTOF3D
MOVJ C00182 BC00182 VJ=100.00  +MOVJ EC00182 VJ=100.00
MOVL C00183 BC00183 V=400.0  +MOVJ EC00183 VJ=100.00
SMOVL C00184 BC00184 V=100.0  +MOVJ EC00184
SREFP 3 C00185 BC00185  +REFP EC00185
CALL JOB:SEARCH-R1-S13D
SET P041 P006
SFTON3D P041
SMOVL C00186 BC00186 V=100.0  +MOVJ EC00186
SREFP 3 C00187 BC00187  +REFP EC00187
CALL JOB:SEARCH-R1-S13D
SET P041 P006
SFTON3D P041
SMOVL C00188 BC00188 V=100.0  +MOVJ EC00188
SREFP 3 C00189 BC00189  +REFP EC00189
CALL JOB:SEARCH-R1-S13D
SET P041 P006
SFTON3D P041
SMOVL C00190 BC00190 V=100.0  +MOVJ EC00190
MOVL C00191 BC00191 V=400.0  +MOVJ EC00191 VJ=100.00
MOVL C00192 BC00192 V=1000.0  +MOVJ EC00192 VJ=100.00
'Path W3545
SFTOF3D
SFTON3D P041
MOVJ C00193 BC00193 VJ=100.00  +MOVJ EC00193 VJ=100.00
SMOVL C00194 BC00194 V=400.0  +MOVJ EC00194
SMOVL C00195 BC00195 V=133.3 PL=0  +MOVJ EC00195
SREFP 1 C00196 BC00196  +REFP EC00196
SREFP 2 C00197 BC00197  +REFP EC00197
MACRO1 MJ#(0) ARGF9
ARCON
SWVON WEV#(61)
SMOVL C00198 BC00198 V=6.7  +MOVJ EC00198
SMOVL C00199 BC00199 V=6.7  +MOVJ EC00199
SMOVL C00200 BC00200 V=6.7  +MOVJ EC00200
ARCOF
SWVOF
SMOVL C00201 BC00201 V=400.0  +MOVJ EC00201
SMOVL C00202 BC00202 V=1000.0  +MOVJ EC00202
SFTOF3D
'Path W3546
SFTOF3D
SFTON3D P042
MOVJ C00203 BC00203 VJ=100.00  +MOVJ EC00203 VJ=100.00
MOVJ C00204 BC00204 VJ=100.00  +MOVJ EC00204 VJ=100.00
SMOVL C00205 BC00205 V=400.0  +MOVJ EC00205
SMOVL C00206 BC00206 V=133.3 PL=0  +MOVJ EC00206
SREFP 1 C00207 BC00207  +REFP EC00207
SREFP 2 C00208 BC00208  +REFP EC00208
MACRO1 MJ#(0) ARGF14
ARCON
SMOVL C00209 BC00209 V=8.3  +MOVJ EC00209
SMOVL C00210 BC00210 V=8.3  +MOVJ EC00210
SMOVL C00211 BC00211 V=8.3  +MOVJ EC00211
ARCOF
SMOVL C00212 BC00212 V=400.0  +MOVJ EC00212
SMOVL C00213 BC00213 V=333.3  +MOVJ EC00213
SFTOF3D
MOVJ C00214 BC00214 VJ=100.00  +MOVJ EC00214 VJ=100.00
'Path W3547
SFTOF3D
SFTON3D P043
MOVJ C00215 BC00215 VJ=100.00  +MOVJ EC00215 VJ=100.00
MOVJ C00216 BC00216 VJ=100.00  +MOVJ EC00216 VJ=100.00
SMOVL C00217 BC00217 V=400.0  +MOVJ EC00217
SMOVL C00218 BC00218 V=133.3 PL=0  +MOVJ EC00218
SREFP 1 C00219 BC00219  +REFP EC00219
SREFP 2 C00220 BC00220  +REFP EC00220
MACRO1 MJ#(0) ARGF14
ARCON
SMOVL C00221 BC00221 V=8.3  +MOVJ EC00221
SMOVL C00222 BC00222 V=8.3  +MOVJ EC00222
ARCOF
SMOVL C00223 BC00223 V=400.0  +MOVJ EC00223
SMOVL C00224 BC00224 V=1000.0  +MOVJ EC00224
SMOVL C00225 BC00225 V=1000.0  +MOVJ EC00225
SFTOF3D
'NIE SPAWAMY
COMM 'Path W3548
COMM SFTOF3D
COMM SFTON3D P044
COMM MOVJ C00226 BC00226 VJ=100.00  +MOVJ EC00226 VJ=100.00
COMM SMOVL C00227 BC00227 V=400.0  +MOVJ EC00227
COMM SMOVL C00228 BC00228 V=100.0 PL=0  +MOVJ EC00228
COMM SREFP 1 C00229 BC00229  +REFP EC00229
COMM SREFP 2 C00230 BC00230  +REFP EC00230
COMM MACRO1 MJ#(0) ARGF0
COMM ARCON
COMM SMOVL C00231 BC00231 V=10.0  +MOVJ EC00231
COMM SMOVL C00232 BC00232 V=10.0  +MOVJ EC00232
COMM SMOVL C00233 BC00233 V=10.0  +MOVJ EC00233
COMM SMOVL C00234 BC00234 V=10.0  +MOVJ EC00234
COMM SMOVL C00235 BC00235 V=10.0  +MOVJ EC00235
COMM SMOVL C00236 BC00236 V=10.0  +MOVJ EC00236
COMM SMOVL C00237 BC00237 V=10.0  +MOVJ EC00237
COMM SMOVL C00238 BC00238 V=10.0  +MOVJ EC00238
COMM SMOVL C00239 BC00239 V=10.0  +MOVJ EC00239
COMM SMOVL C00240 BC00240 V=10.0  +MOVJ EC00240
COMM SMOVL C00241 BC00241 V=10.0  +MOVJ EC00241
COMM SMOVL C00242 BC00242 V=10.0  +MOVJ EC00242
COMM SMOVL C00243 BC00243 V=10.0  +MOVJ EC00243
COMM SMOVL C00244 BC00244 V=10.0  +MOVJ EC00244
COMM SMOVL C00245 BC00245 V=10.0  +MOVJ EC00245
COMM SMOVL C00246 BC00246 V=10.0  +MOVJ EC00246
COMM SMOVL C00247 BC00247 V=10.0  +MOVJ EC00247
COMM SMOVL C00248 BC00248 V=10.0  +MOVJ EC00248
COMM SMOVL C00249 BC00249 V=10.0  +MOVJ EC00249
COMM SMOVL C00250 BC00250 V=10.0  +MOVJ EC00250
COMM SMOVL C00251 BC00251 V=10.0  +MOVJ EC00251
COMM SMOVL C00252 BC00252 V=10.0  +MOVJ EC00252
COMM SMOVL C00253 BC00253 V=10.0  +MOVJ EC00253
COMM SMOVL C00254 BC00254 V=10.0  +MOVJ EC00254
COMM SMOVL C00255 BC00255 V=10.0  +MOVJ EC00255
COMM ARCOF
COMM SMOVL C00256 BC00256 V=400.0  +MOVJ EC00256
COMM SMOVL C00257 BC00257 V=1000.0  +MOVJ EC00257
COMM SFTOF3D
'Path W3549
SFTOF3D
MOVJ C00258 BC00258 VJ=100.00  +MOVJ EC00258 VJ=100.00
MOVJ C00259 BC00259 VJ=100.00  +MOVJ EC00259 VJ=100.00
SFTON3D P045
MOVJ C00260 BC00260 VJ=100.00  +MOVJ EC00260 VJ=100.00
SMOVL C00261 BC00261 V=400.0  +MOVJ EC00261
SMOVL C00262 BC00262 V=100.0 PL=0  +MOVJ EC00262
SREFP 1 C00263 BC00263  +REFP EC00263
SREFP 2 C00264 BC00264  +REFP EC00264
MACRO1 MJ#(0) ARGF14
ARCON
SMOVL C00265 BC00265 V=8.3  +MOVJ EC00265
SMOVL C00266 BC00266 V=8.3  +MOVJ EC00266
SMOVL C00267 BC00267 V=8.3  +MOVJ EC00267
SMOVL C00268 BC00268 V=8.3  +MOVJ EC00268
SMOVL C00269 BC00269 V=8.3  +MOVJ EC00269
ARCOF
SMOVL C00270 BC00270 V=400.0  +MOVJ EC00270
SMOVL C00271 BC00271 V=1000.0  +MOVJ EC00271
SMOVL C00272 BC00272 V=1000.0  +MOVJ EC00272
MOVJ C00273 BC00273 VJ=100.00  +MOVJ EC00273 VJ=50.00
SFTOF3D
'Path W3550
SFTOF3D
SFTON3D P046
MOVJ C00274 BC00274 VJ=100.00  +MOVJ EC00274 VJ=100.00
MOVJ C00275 BC00275 VJ=100.00  +MOVJ EC00275 VJ=100.00
SMOVL C00276 BC00276 V=400.0  +MOVJ EC00276
SMOVL C00277 BC00277 V=100.0 PL=0  +MOVJ EC00277
SREFP 1 C00278 BC00278  +REFP EC00278
SREFP 2 C00279 BC00279  +REFP EC00279
MACRO1 MJ#(0) ARGF14
ARCON
SMOVL C00280 BC00280 V=8.3  +MOVJ EC00280
SMOVL C00281 BC00281 V=8.3  +MOVJ EC00281
SMOVL C00282 BC00282 V=8.3  +MOVJ EC00282
SMOVL C00283 BC00283 V=8.3  +MOVJ EC00283
SMOVL C00284 BC00284 V=8.3  +MOVJ EC00284
SMOVL C00285 BC00285 V=8.3  +MOVJ EC00285
ARCOF
SMOVL C00286 BC00286 V=400.0  +MOVJ EC00286
SMOVL C00287 BC00287 V=1000.0  +MOVJ EC00287
SFTOF3D
MOVJ C00288 BC00288 VJ=100.00  +MOVJ EC00288 VJ=100.00
MOVJ C00289 BC00289 VJ=100.00  +MOVJ EC00289 VJ=100.00
MOVJ C00290 BC00290 VJ=100.00  +MOVJ EC00290 VJ=100.00
'Down
'Path W3551
SFTOF3D
MOVJ C00291 BC00291 VJ=100.00  +MOVJ EC00291 VJ=100.00
MOVL C00292 BC00292 V=400.0  +MOVJ EC00292 VJ=100.00
SFTON3D P032
SMOVL C00293 BC00293 V=100.0 PL=0  +MOVJ EC00293
SREFP 1 C00294 BC00294  +REFP EC00294
SREFP 2 C00295 BC00295  +REFP EC00295
MACRO1 MJ#(0) ARGF21
ARCON
SWVON WEV#(100)
SMOVC C00296 BC00296 V=9.2  +MOVJ EC00296
SMOVC C00297 BC00297 V=9.2  +MOVJ EC00297
SMOVC C00298 BC00298 V=9.2  +MOVJ EC00298
SMOVC C00299 BC00299 V=9.2  +MOVJ EC00299
SMOVC C00300 BC00300 V=9.2  +MOVJ EC00300
ARCOF
SFTOF3D
SWVOF
MOVL C00301 BC00301 V=400.0  +MOVJ EC00301 VJ=100.00
MOVL C00302 BC00302 V=1000.0  +MOVJ EC00302 VJ=100.00
MOVJ C00303 BC00303 VJ=100.00  +MOVJ EC00303 VJ=100.00
MOVJ C00304 BC00304 VJ=100.00  +MOVJ EC00304 VJ=100.00
MOVJ C00305 BC00305 VJ=100.00  +MOVJ EC00305 VJ=100.00
'Path W3552
SFTOF3D
COMM PAUSE
COMM SFTON3D P022
COMM MOVJ C00306 BC00306 VJ=100.00  +MOVJ EC00306 VJ=100.00
COMM SMOVL C00307 BC00307 V=333.3  +MOVJ EC00307
COMM SMOVL C00308 BC00308 V=133.3 PL=0  +MOVJ EC00308
COMM SREFP 1 C00309 BC00309  +REFP EC00309
COMM SREFP 2 C00310 BC00310  +REFP EC00310
COMM MACRO1 MJ#(0) ARGF14
COMM ARCON
COMM SMOVC C00311 BC00311 V=8.3  +MOVJ EC00311
COMM SMOVC C00312 BC00312 V=8.3  +MOVJ EC00312
COMM SMOVC C00313 BC00313 V=8.3  +MOVJ EC00313
COMM SMOVC C00314 BC00314 V=8.3  +MOVJ EC00314
COMM SMOVC C00315 BC00315 V=8.3  +MOVJ EC00315
COMM SMOVC C00316 BC00316 V=8.3  +MOVJ EC00316
COMM SMOVL C00317 BC00317 V=8.3  +MOVJ EC00317
COMM ARCOF
COMM SMOVL C00318 BC00318 V=400.0  +MOVJ EC00318
COMM SMOVL C00319 BC00319 V=1000.0  +MOVJ EC00319
COMM SFTOF3D
COMM 'Path W3553
COMM SFTOF3D
COMM SFTON3D P022
COMM MOVJ C00320 BC00320 VJ=100.00  +MOVJ EC00320 VJ=100.00
COMM SMOVL C00321 BC00321 V=133.3  +MOVJ EC00321
COMM 'SZEROKA SZCZELINA!!!
COMM MACRO1 MJ#(0) ARGF14
COMM SMOVL C00322 BC00322 V=133.3 PL=0  +MOVJ EC00322
COMM SREFP 1 C00323 BC00323  +REFP EC00323
COMM SREFP 2 C00324 BC00324  +REFP EC00324
COMM ARCON
COMM SWVON WEV#(14)
COMM SMOVL C00325 BC00325 V=7.5  +MOVJ EC00325
COMM SMOVL C00326 BC00326 V=7.5  +MOVJ EC00326
COMM ARCOF
COMM SWVOF
COMM SMOVL C00327 BC00327 V=400.0  +MOVJ EC00327
COMM SFTOF3D
SMOVL C00328 BC00328 V=1000.0  +MOVJ EC00328
MOVJ C00329 BC00329 VJ=70.00  +MOVJ EC00329 VJ=70.00
MACRO1 MJ#(0) ARGF14
SFTON3D P088
SMOVL C00330 BC00330 V=166.7  +MOVJ EC00330
ARCON
SMOVL C00331 BC00331 V=10.8  +MOVJ EC00331
ARCOF
SFTOF3D
SMOVL C00332 BC00332 V=250.0  +MOVJ EC00332
'
'NIE SPAWAMY_BRAK BLASZKI
COMM 'Path W3554
COMM SFTOF3D
COMM SFTON3D P023
COMM MOVJ C00333 BC00333 VJ=100.00  +MOVJ EC00333 VJ=100.00
COMM MOVJ C00334 BC00334 VJ=100.00  +MOVJ EC00334 VJ=100.00
COMM SMOVL C00335 BC00335 V=400.0  +MOVJ EC00335
COMM SMOVL C00336 BC00336 V=100.0 PL=0  +MOVJ EC00336
COMM SREFP 1 C00337 BC00337  +REFP EC00337
COMM SREFP 2 C00338 BC00338  +REFP EC00338
COMM MACRO1 MJ#(0) ARGF0
COMM ARCON
COMM SMOVL C00339 BC00339 V=10.0  +MOVJ EC00339
COMM SMOVL C00340 BC00340 V=10.0  +MOVJ EC00340
COMM SMOVL C00341 BC00341 V=10.0  +MOVJ EC00341
COMM ARCOF
COMM SMOVL C00342 BC00342 V=400.0  +MOVJ EC00342
COMM SMOVL C00343 BC00343 V=1000.0  +MOVJ EC00343
COMM SFTOF3D
COMM MOVJ C00344 BC00344 VJ=100.00  +MOVJ EC00344 VJ=100.00
'NIE SPAWAMY_BRAK BLASZKI
COMM 'Path W3555
COMM SFTOF3D
COMM SFTON3D P023
COMM MOVJ C00345 BC00345 VJ=100.00  +MOVJ EC00345 VJ=100.00
COMM SMOVL C00346 BC00346 V=100.0  +MOVJ EC00346
COMM SMOVL C00347 BC00347 V=100.0 PL=0  +MOVJ EC00347
COMM SREFP 1 C00348 BC00348  +REFP EC00348
COMM SREFP 2 C00349 BC00349  +REFP EC00349
COMM MACRO1 MJ#(0) ARGF0
COMM ARCON
COMM SMOVL C00350 BC00350 V=10.0  +MOVJ EC00350
COMM SMOVL C00351 BC00351 V=10.0  +MOVJ EC00351
COMM SMOVL C00352 BC00352 V=10.0  +MOVJ EC00352
COMM ARCOF
COMM SMOVL C00353 BC00353 V=400.0  +MOVJ EC00353
COMM SMOVL C00354 BC00354 V=1000.0  +MOVJ EC00354
COMM SMOVL C00355 BC00355 V=1000.0  +MOVJ EC00355
COMM SFTOF3D
'NIE SPAWAMY_BRAK BLASZKI
COMM 'Path W3556
COMM SFTOF3D
COMM SFTON3D P023
COMM MOVJ C00356 BC00356 VJ=100.00  +MOVJ EC00356 VJ=100.00
COMM SMOVL C00357 BC00357 V=100.0  +MOVJ EC00357
COMM SMOVL C00358 BC00358 V=100.0 PL=0  +MOVJ EC00358
COMM SREFP 1 C00359 BC00359  +REFP EC00359
COMM SREFP 2 C00360 BC00360  +REFP EC00360
COMM MACRO1 MJ#(0) ARGF0
COMM ARCON
COMM SMOVL C00361 BC00361 V=10.0  +MOVJ EC00361
COMM ARCOF
COMM SMOVL C00362 BC00362 V=400.0  +MOVJ EC00362
COMM SMOVL C00363 BC00363 V=1000.0  +MOVJ EC00363
COMM SFTOF3D
'
'NIE SPAWAMY_BRAK BLASZKI
COMM 'Path W3557
COMM SFTOF3D
COMM SFTON3D P024
COMM MOVJ C00364 BC00364 VJ=100.00  +MOVJ EC00364 VJ=100.00
COMM SMOVL C00365 BC00365 V=100.0  +MOVJ EC00365
COMM SMOVL C00366 BC00366 V=100.0 PL=0  +MOVJ EC00366
COMM SREFP 1 C00367 BC00367  +REFP EC00367
COMM SREFP 2 C00368 BC00368  +REFP EC00368
COMM MACRO1 MJ#(0) ARGF0
COMM ARCON
COMM SMOVL C00369 BC00369 V=10.0  +MOVJ EC00369
COMM SMOVL C00370 BC00370 V=10.0  +MOVJ EC00370
COMM SMOVL C00371 BC00371 V=10.0  +MOVJ EC00371
COMM ARCOF
COMM SMOVL C00372 BC00372 V=400.0  +MOVJ EC00372
COMM SMOVL C00373 BC00373 V=1000.0  +MOVJ EC00373
COMM SFTOF3D
COMM MOVJ C00374 BC00374 VJ=100.00  +MOVJ EC00374 VJ=100.00
'NIE SPAWAMY_BRAK BLASZKI
COMM 'Path W3558
COMM SFTOF3D
COMM SFTON3D P024
COMM MOVJ C00375 BC00375 VJ=100.00  +MOVJ EC00375 VJ=100.00
COMM SMOVL C00376 BC00376 V=100.0  +MOVJ EC00376
COMM SMOVL C00377 BC00377 V=100.0 PL=0  +MOVJ EC00377
COMM SREFP 1 C00378 BC00378  +REFP EC00378
COMM SREFP 2 C00379 BC00379  +REFP EC00379
COMM MACRO1 MJ#(0) ARGF0
COMM ARCON
COMM SMOVL C00380 BC00380 V=10.0  +MOVJ EC00380
COMM SMOVL C00381 BC00381 V=10.0  +MOVJ EC00381
COMM SMOVL C00382 BC00382 V=10.0  +MOVJ EC00382
COMM ARCOF
COMM SMOVL C00383 BC00383 V=400.0  +MOVJ EC00383
COMM SMOVL C00384 BC00384 V=1000.0  +MOVJ EC00384
COMM SMOVL C00385 BC00385 V=1000.0  +MOVJ EC00385
COMM SFTOF3D
'NIE SPAWAMY_BRAK BLASZKI
COMM 'Path W3559
COMM SFTOF3D
COMM SFTON3D P024
COMM MOVJ C00386 BC00386 VJ=100.00  +MOVJ EC00386 VJ=100.00
COMM SMOVL C00387 BC00387 V=100.0  +MOVJ EC00387
COMM SMOVL C00388 BC00388 V=100.0 PL=0  +MOVJ EC00388
COMM SREFP 1 C00389 BC00389  +REFP EC00389
COMM SREFP 2 C00390 BC00390  +REFP EC00390
COMM MACRO1 MJ#(0) ARGF0
COMM ARCON
COMM SMOVL C00391 BC00391 V=10.0  +MOVJ EC00391
COMM ARCOF
COMM SMOVL C00392 BC00392 V=400.0  +MOVJ EC00392
COMM SMOVL C00393 BC00393 V=1000.0  +MOVJ EC00393
COMM SFTOF3D
COMM MOVJ C00394 BC00394 VJ=100.00  +MOVJ EC00394 VJ=100.00
'
'NIE SPAWAMY_BRAK BLASZKI
COMM 'Path W3560
COMM SFTOF3D
COMM SFTON3D P025
COMM MOVJ C00395 BC00395 VJ=100.00  +MOVJ EC00395 VJ=100.00
COMM SMOVL C00396 BC00396 V=100.0  +MOVJ EC00396
COMM SMOVL C00397 BC00397 V=100.0 PL=0  +MOVJ EC00397
COMM SREFP 1 C00398 BC00398  +REFP EC00398
COMM SREFP 2 C00399 BC00399  +REFP EC00399
COMM MACRO1 MJ#(0) ARGF0
COMM ARCON
COMM SMOVL C00400 BC00400 V=10.0  +MOVJ EC00400
COMM SMOVL C00401 BC00401 V=10.0  +MOVJ EC00401
COMM SMOVL C00402 BC00402 V=10.0  +MOVJ EC00402
COMM ARCOF
COMM SMOVL C00403 BC00403 V=400.0  +MOVJ EC00403
COMM SMOVL C00404 BC00404 V=1000.0  +MOVJ EC00404
COMM SFTOF3D
COMM MOVJ C00405 BC00405 VJ=100.00  +MOVJ EC00405 VJ=100.00
'NIE SPAWAMY_BRAK BLASZKI
COMM 'Path W3561
COMM SFTOF3D
COMM SFTON3D P025
COMM MOVJ C00406 BC00406 VJ=100.00  +MOVJ EC00406 VJ=100.00
COMM SMOVL C00407 BC00407 V=100.0  +MOVJ EC00407
COMM SMOVL C00408 BC00408 V=100.0 PL=0  +MOVJ EC00408
COMM SREFP 1 C00409 BC00409  +REFP EC00409
COMM SREFP 2 C00410 BC00410  +REFP EC00410
COMM MACRO1 MJ#(0) ARGF0
COMM ARCON
COMM SMOVL C00411 BC00411 V=10.0  +MOVJ EC00411
COMM SMOVL C00412 BC00412 V=10.0  +MOVJ EC00412
COMM SMOVL C00413 BC00413 V=10.0  +MOVJ EC00413
COMM ARCOF
COMM SMOVL C00414 BC00414 V=400.0  +MOVJ EC00414
COMM SMOVL C00415 BC00415 V=1000.0  +MOVJ EC00415
COMM SMOVL C00416 BC00416 V=1000.0  +MOVJ EC00416
COMM SFTOF3D
'NIE SPAWAMY_BRAK BLASZKI
COMM 'Path W3562
COMM SFTOF3D
COMM SFTON3D P025
COMM MOVJ C00417 BC00417 VJ=100.00  +MOVJ EC00417 VJ=100.00
COMM SMOVL C00418 BC00418 V=100.0  +MOVJ EC00418
COMM SMOVL C00419 BC00419 V=100.0 PL=0  +MOVJ EC00419
COMM SREFP 1 C00420 BC00420  +REFP EC00420
COMM SREFP 2 C00421 BC00421  +REFP EC00421
COMM MACRO1 MJ#(0) ARGF0
COMM ARCON
COMM SMOVL C00422 BC00422 V=10.0  +MOVJ EC00422
COMM ARCOF
COMM SMOVL C00423 BC00423 V=400.0  +MOVJ EC00423
COMM SMOVL C00424 BC00424 V=1000.0  +MOVJ EC00424
COMM SFTOF3D
COMM MOVJ C00425 BC00425 VJ=100.00  +MOVJ EC00425 VJ=100.00
COMM MOVJ C00426 BC00426 VJ=100.00  +MOVJ EC00426 VJ=100.00
COMM '
COMM MOVJ C00427 BC00427 VJ=100.00  +MOVJ EC00427 VJ=100.00
COMM MOVJ C00428 BC00428 VJ=100.00  +MOVJ EC00428 VJ=100.00
'NIE SPAWAMY_BRAK BLASZKI
COMM 'Path W3563
COMM SFTOF3D
COMM SFTON3D P023
COMM MOVJ C00429 BC00429 VJ=100.00  +MOVJ EC00429 VJ=100.00
COMM SMOVL C00430 BC00430 V=400.0  +MOVJ EC00430
COMM SMOVL C00431 BC00431 V=100.0 PL=0  +MOVJ EC00431
COMM SREFP 1 C00432 BC00432  +REFP EC00432
COMM SREFP 2 C00433 BC00433  +REFP EC00433
COMM MACRO1 MJ#(0) ARGF0
COMM ARCON
COMM SMOVL C00434 BC00434 V=10.0  +MOVJ EC00434
COMM SMOVL C00435 BC00435 V=10.0  +MOVJ EC00435
COMM SMOVL C00436 BC00436 V=10.0  +MOVJ EC00436
COMM ARCOF
COMM SMOVL C00437 BC00437 V=400.0  +MOVJ EC00437
COMM SMOVL C00438 BC00438 V=1000.0  +MOVJ EC00438
COMM SMOVL C00439 BC00439 V=1000.0  +MOVJ EC00439
COMM SFTOF3D
'NIE SPAWAMY_BRAK BLASZKI
COMM 'Path W3564
COMM SFTOF3D
COMM SFTON3D P023
COMM SMOVL C00440 BC00440 V=100.0  +MOVJ EC00440
COMM SMOVL C00441 BC00441 V=100.0 PL=0  +MOVJ EC00441
COMM SREFP 1 C00442 BC00442  +REFP EC00442
COMM SREFP 2 C00443 BC00443  +REFP EC00443
COMM MACRO1 MJ#(0) ARGF0
COMM ARCON
COMM SMOVL C00444 BC00444 V=10.0  +MOVJ EC00444
COMM SMOVL C00445 BC00445 V=10.0  +MOVJ EC00445
COMM SMOVL C00446 BC00446 V=10.0  +MOVJ EC00446
COMM ARCOF
COMM SMOVL C00447 BC00447 V=400.0  +MOVJ EC00447
COMM SFTOF3D
COMM MOVJ C00448 BC00448 VJ=100.00  +MOVJ EC00448 VJ=100.00
'
COMM MOVJ C00449 BC00449 VJ=100.00  +MOVJ EC00449 VJ=100.00
'NIE SPAWAMY_BRAK BLASZKI
COMM 'Path W3565
COMM SFTOF3D
COMM SFTON3D P024
COMM MOVJ C00450 BC00450 VJ=100.00  +MOVJ EC00450 VJ=100.00
COMM MOVJ C00451 BC00451 VJ=100.00  +MOVJ EC00451 VJ=100.00
COMM SMOVL C00452 BC00452 V=400.0  +MOVJ EC00452
COMM SMOVL C00453 BC00453 V=100.0 PL=0  +MOVJ EC00453
COMM SREFP 1 C00454 BC00454  +REFP EC00454
COMM SREFP 2 C00455 BC00455  +REFP EC00455
COMM MACRO1 MJ#(0) ARGF0
COMM ARCON
COMM SMOVL C00456 BC00456 V=10.0  +MOVJ EC00456
COMM SMOVL C00457 BC00457 V=10.0  +MOVJ EC00457
COMM SMOVL C00458 BC00458 V=10.0  +MOVJ EC00458
COMM ARCOF
COMM SMOVL C00459 BC00459 V=400.0  +MOVJ EC00459
COMM SMOVL C00460 BC00460 V=1000.0  +MOVJ EC00460
COMM SMOVL C00461 BC00461 V=1000.0  +MOVJ EC00461
COMM SFTOF3D
'NIE SPAWAMY_BRAK BLASZKI
COMM 'Path W3566
COMM SFTOF3D
COMM SFTON3D P025
COMM MOVJ C00462 BC00462 VJ=100.00  +MOVJ EC00462 VJ=100.00
COMM SMOVL C00463 BC00463 V=400.0  +MOVJ EC00463
COMM SMOVL C00464 BC00464 V=100.0 PL=0  +MOVJ EC00464
COMM SREFP 1 C00465 BC00465  +REFP EC00465
COMM SREFP 2 C00466 BC00466  +REFP EC00466
COMM MACRO1 MJ#(0) ARGF0
COMM ARCON
COMM SMOVL C00467 BC00467 V=10.0  +MOVJ EC00467
COMM SMOVL C00468 BC00468 V=10.0  +MOVJ EC00468
COMM SMOVL C00469 BC00469 V=10.0  +MOVJ EC00469
COMM ARCOF
COMM SMOVL C00470 BC00470 V=400.0  +MOVJ EC00470
COMM SMOVL C00471 BC00471 V=1000.0  +MOVJ EC00471
COMM SMOVL C00472 BC00472 V=1000.0  +MOVJ EC00472
COMM SFTOF3D
MOVJ C00473 BC00473 VJ=100.00  +MOVJ EC00473 VJ=100.00
MOVJ C00474 BC00474 VJ=100.00  +MOVJ EC00474 VJ=50.00
MOVJ C00475 BC00475 VJ=100.00  +MOVJ EC00475 VJ=50.00
MOVJ C00476 BC00476 VJ=100.00  +MOVJ EC00476 VJ=50.00
MOVJ C00477 BC00477 VJ=100.00  +MOVJ EC00477 VJ=100.00
'Path W3567
SFTOF3D
SFTON3D P021
MOVJ C00478 BC00478 VJ=100.00  +MOVJ EC00478 VJ=100.00
SMOVL C00479 BC00479 V=250.0  +MOVJ EC00479
SMOVL C00480 BC00480 V=133.3 PL=0  +MOVJ EC00480
SREFP 1 C00481 BC00481  +REFP EC00481
SREFP 2 C00482 BC00482  +REFP EC00482
MACRO1 MJ#(0) ARGF21
ARCON
SWVON WEV#(100)
SMOVC C00483 BC00483 V=9.2  +MOVJ EC00483
SMOVC C00484 BC00484 V=9.2  +MOVJ EC00484
SMOVC C00485 BC00485 V=9.2  +MOVJ EC00485
SMOVC C00486 BC00486 V=9.2  +MOVJ EC00486
ARCOF
SWVOF
SMOVL C00487 BC00487 V=400.0  +MOVJ EC00487
SMOVL C00488 BC00488 V=1000.0  +MOVJ EC00488
SFTOF3D
MOVJ C00489 BC00489 VJ=100.00  +MOVJ EC00489 VJ=100.00
'
MOVJ C00490 BC00490 VJ=100.00  +MOVJ EC00490 VJ=100.00
MOVJ C00491 BC00491 VJ=100.00  +MOVJ EC00491 VJ=100.00
'NIE SPAWAMY_BRAK BLASZKI
COMM 'Path W3568
COMM SFTOF3D
COMM SFTON3D P024
COMM MOVJ C00492 BC00492 VJ=100.00  +MOVJ EC00492 VJ=100.00
COMM SMOVL C00493 BC00493 V=100.0  +MOVJ EC00493
COMM SMOVL C00494 BC00494 V=100.0 PL=0  +MOVJ EC00494
COMM SREFP 1 C00495 BC00495  +REFP EC00495
COMM SREFP 2 C00496 BC00496  +REFP EC00496
COMM MACRO1 MJ#(0) ARGF0
COMM ARCON
COMM SMOVL C00497 BC00497 V=10.0  +MOVJ EC00497
COMM SMOVL C00498 BC00498 V=10.0  +MOVJ EC00498
COMM SMOVL C00499 BC00499 V=10.0  +MOVJ EC00499
COMM ARCOF
COMM SMOVL C00500 BC00500 V=400.0  +MOVJ EC00500
COMM SMOVL C00501 BC00501 V=1000.0  +MOVJ EC00501
COMM SFTOF3D
'NIE SPAWAMY_BRAK BLASZKI
COMM 'Path W3569
COMM SFTOF3D
COMM SFTON3D P025
COMM MOVJ C00502 BC00502 VJ=100.00  +MOVJ EC00502 VJ=100.00
COMM SMOVL C00503 BC00503 V=100.0  +MOVJ EC00503
COMM SMOVL C00504 BC00504 V=100.0 PL=0  +MOVJ EC00504
COMM SREFP 1 C00505 BC00505  +REFP EC00505
COMM SREFP 2 C00506 BC00506  +REFP EC00506
COMM MACRO1 MJ#(0) ARGF0
COMM ARCON
COMM SMOVL C00507 BC00507 V=10.0  +MOVJ EC00507
COMM SMOVL C00508 BC00508 V=10.0  +MOVJ EC00508
COMM SMOVL C00509 BC00509 V=10.0  +MOVJ EC00509
COMM ARCOF
COMM SMOVL C00510 BC00510 V=400.0  +MOVJ EC00510
COMM SMOVL C00511 BC00511 V=1000.0  +MOVJ EC00511
COMM SMOVL C00512 BC00512 V=1000.0  +MOVJ EC00512
COMM SFTOF3D
COMM MOVJ C00513 BC00513 VJ=100.00  +MOVJ EC00513 VJ=100.00
COMM '
COMM MOVJ C00514 BC00514 VJ=100.00  +MOVJ EC00514 VJ=100.00
COMM MOVJ C00515 BC00515 VJ=100.00  +MOVJ EC00515 VJ=100.00
'Path W3570
SFTOF3D
SFTON3D P026
MOVJ C00516 BC00516 VJ=100.00  +MOVJ EC00516 VJ=100.00
MOVJ C00517 BC00517 VJ=100.00  +MOVJ EC00517 VJ=100.00
SMOVL C00518 BC00518 V=666.7  +MOVJ EC00518
SMOVL C00519 BC00519 V=133.3  +MOVJ EC00519
SREFP 1 C00520 BC00520  +REFP EC00520
SREFP 2 C00521 BC00521  +REFP EC00521
MACRO1 MJ#(0) ARGF21
ARCON
SMOVL C00522 BC00522 V=7.5  +MOVJ EC00522
SMOVL C00523 BC00523 V=7.5  +MOVJ EC00523
SMOVL C00524 BC00524 V=7.5  +MOVJ EC00524
SMOVL C00525 BC00525 V=7.5  +MOVJ EC00525
SMOVL C00526 BC00526 V=7.5  +MOVJ EC00526
SMOVL C00527 BC00527 V=7.5  +MOVJ EC00527
SMOVL C00528 BC00528 V=7.5  +MOVJ EC00528
ARCON
SMOVL C00529 BC00529 V=7.5  +MOVJ EC00529
SMOVL C00530 BC00530 V=7.5  +MOVJ EC00530
SMOVL C00531 BC00531 V=7.5  +MOVJ EC00531
SMOVL C00532 BC00532 V=7.5  +MOVJ EC00532
ARCOF
SMOVL C00533 BC00533 V=250.0  +MOVJ EC00533
SMOVL C00534 BC00534 V=1000.0  +MOVJ EC00534
SFTOF3D
MOVJ C00535 BC00535 VJ=100.00  +MOVJ EC00535 VJ=100.00
'jakie searche do takicj spoin?
MOVJ C00536 BC00536 VJ=100.00  +MOVJ EC00536 VJ=100.00
MOVJ C00537 BC00537 VJ=100.00  +MOVJ EC00537 VJ=100.00
'Path W3572
SFTOF3D
'jakie searche do takicj spoin?
MOVJ C00538 BC00538 VJ=100.00  +MOVJ EC00538 VJ=100.00
'Path W3579
SFTOF3D
MOVJ C00539 BC00539 VJ=50.00  +MOVJ EC00539 VJ=100.00
COMM PAUSE
COMM MOVL C00540 BC00540 V=400.0  +MOVJ EC00540 VJ=100.00
COMM SFTOF3D
COMM SFTON3D P089
COMM SMOVL C00541 BC00541 V=100.0 PL=0  +MOVJ EC00541
COMM SREFP 1 C00542 BC00542  +REFP EC00542
COMM SREFP 2 C00543 BC00543  +REFP EC00543
COMM MACRO1 MJ#(0) ARGF9
COMM ARCON
COMM SMOVL C00544 BC00544 V=11.7  +MOVJ EC00544
COMM ARCOF
COMM MOVL C00545 BC00545 V=666.7  +MOVJ EC00545 VJ=100.00
COMM SMOVL C00546 BC00546 V=166.7  +MOVJ EC00546
COMM ARCON
COMM SMOVL C00547 BC00547 V=11.7  +MOVJ EC00547
COMM ARCOF
COMM SFTOF3D
SMOVL C00548 BC00548 V=250.0  +MOVJ EC00548
MOVJ C00549 BC00549 VJ=100.00  +MOVJ EC00549 VJ=0.78
MACRO1 MJ#(0) ARGF9
MOVL C00550 BC00550 V=1000.0  +MOVJ EC00550 VJ=100.00
SFTON3D P031
SMOVL C00551 BC00551 V=166.7 PL=0  +MOVJ EC00551
ARCON
SMOVL C00552 BC00552 V=13.3  +MOVJ EC00552
SMOVC C00553 BC00553 V=15.0  +MOVJ EC00553
SMOVC C00554 BC00554 V=15.0  +MOVJ EC00554
SMOVC C00555 BC00555 V=15.0  +MOVJ EC00555
SMOVL C00556 BC00556 V=6.7  +MOVJ EC00556
SMOVL C00557 BC00557 V=12.5  +MOVJ EC00557
SFTON3D P032
SMOVL C00558 BC00558 V=12.5  +MOVJ EC00558
ARCOF
SMOVL C00559 BC00559 V=166.7  +MOVJ EC00559
SFTOF3D
MOVL C00560 BC00560 V=1000.0  +MOVJ EC00560 VJ=100.00
SFTON3D P034
SMOVL C00561 BC00561 V=166.7 PL=0  +MOVJ EC00561
ARCON
SMOVL C00562 BC00562 V=13.3  +MOVJ EC00562
SMOVL C00563 BC00563 V=13.3  +MOVJ EC00563
SMOVL C00564 BC00564 V=13.3  +MOVJ EC00564
SMOVL C00565 BC00565 V=13.3  +MOVJ EC00565
SMOVL C00566 BC00566 V=13.3  +MOVJ EC00566
SMOVL C00567 BC00567 V=12.5  +MOVJ EC00567
SFTON3D P033
SMOVL C00568 BC00568 V=12.5  +MOVJ EC00568
ARCOF
SMOVL C00569 BC00569 V=166.7  +MOVJ EC00569
SFTOF3D
MOVL C00570 BC00570 V=1000.0  +MOVJ EC00570 VJ=100.00
SFTON3D P035
SMOVL C00571 BC00571 V=166.7 PL=0  +MOVJ EC00571
ARCON
SMOVL C00572 BC00572 V=13.3  +MOVJ EC00572
SMOVL C00573 BC00573 V=15.0  +MOVJ EC00573
SMOVL C00574 BC00574 V=15.0  +MOVJ EC00574
SMOVL C00575 BC00575 V=12.5  +MOVJ EC00575
SFTON3D P036
SMOVL C00576 BC00576 V=12.5  +MOVJ EC00576
SMOVL C00577 BC00577 V=15.0  +MOVJ EC00577
SMOVL C00578 BC00578 V=15.0  +MOVJ EC00578
ARCOF
SMOVL C00579 BC00579 V=166.7  +MOVJ EC00579
SFTOF3D
SMOVL C00580 BC00580 V=1000.0  +MOVJ EC00580
MACRO1 MJ#(0) ARGF14
MOVL C00581 BC00581 V=1000.0  +MOVJ EC00581 VJ=100.00
SFTON3D P090
SMOVL C00582 BC00582 V=166.7  +MOVJ EC00582
ARCON
SMOVL C00583 BC00583 V=12.5  +MOVJ EC00583
ARCOF
SMOVL C00584 BC00584 V=166.7  +MOVJ EC00584
SMOVL C00585 BC00585 V=166.7  +MOVJ EC00585
SMOVL C00586 BC00586 V=166.7  +MOVJ EC00586
ARCON
SMOVL C00587 BC00587 V=10.8  +MOVJ EC00587
ARCOF
SMOVL C00588 BC00588 V=166.7  +MOVJ EC00588
SFTOF3D
SMOVL C00589 BC00589 V=1000.0  +MOVJ EC00589
MOVJ C00590 BC00590 VJ=100.00  +MOVJ EC00590 VJ=100.00
COMM MOVJ C00591 BC00591 VJ=100.00  +MOVJ EC00591 VJ=100.00
COMM MOVJ C00592 BC00592 VJ=100.00  +MOVJ EC00592 VJ=100.00
'NIE SPAWAMY
COMM 'Path W3582
COMM SFTOF3D
COMM PAUSE
COMM SFTON3D P031
COMM MOVJ C00593 BC00593 VJ=100.00  +MOVJ EC00593 VJ=100.00
COMM SMOVL C00594 BC00594 V=100.0  +MOVJ EC00594
COMM SMOVL C00595 BC00595 V=100.0 PL=0  +MOVJ EC00595
COMM SREFP 1 C00596 BC00596  +REFP EC00596
COMM SREFP 2 C00597 BC00597  +REFP EC00597
COMM MACRO1 MJ#(0) ARGF0
COMM ARCON
COMM SMOVL C00598 BC00598 V=10.0  +MOVJ EC00598
COMM SMOVL C00599 BC00599 V=10.0  +MOVJ EC00599
COMM SMOVL C00600 BC00600 V=10.0  +MOVJ EC00600
COMM ARCOF
COMM SMOVL C00601 BC00601 V=400.0  +MOVJ EC00601
COMM SMOVL C00602 BC00602 V=1000.0  +MOVJ EC00602
COMM SFTOF3D
'Down
MOVJ C00603 BC00603 VJ=100.00  +MOVJ EC00603 VJ=100.00
END
